C01806=1141.439,9.423,-49.221,179.746,6.279,149.212
C01807=1141.445,9.174,-49.208,179.743,6.278,149.213
C01808=1141.450,8.924,-49.194,179.741,6.277,149.213
C01809=1141.455,8.675,-49.181,179.739,6.276,149.214
C01810=1141.460,8.425,-49.167,179.736,6.275,149.214
C01811=1141.465,8.175,-49.153,179.733,6.274,149.215
C01812=1141.470,7.926,-49.140,179.731,6.273,149.215
C01813=1141.475,7.676,-49.126,179.729,6.273,149.216
C01814=1141.480,7.427,-49.113,179.726,6.272,149.216
C01815=1141.485,7.177,-49.100,179.723,6.271,149.217
C01816=1141.491,6.928,-49.086,179.721,6.270,149.217
C01817=1141.495,6.678,-49.073,179.718,6.269,149.218
C01818=1141.501,6.429,-49.059,179.716,6.269,149.219
C01819=1141.506,6.178,-49.045,179.714,6.268,149.219
C01820=1141.511,5.929,-49.033,179.711,6.266,149.220
C01821=1141.516,5.679,-49.018,179.709,6.266,149.220
C01822=1141.522,5.430,-49.006,179.706,6.265,149.221
C01823=1141.526,5.180,-48.991,179.704,6.264,149.221
C01824=1141.532,4.931,-48.979,179.701,6.263,149.222
C01825=1141.537,4.681,-48.965,179.698,6.262,149.223
C01826=1141.542,4.432,-48.951,179.696,6.262,149.223
C01827=1141.547,4.182,-48.938,179.693,6.261,149.224
C01828=1141.552,3.933,-48.924,179.691,6.260,149.224
C01829=1141.557,3.683,-48.911,179.689,6.259,149.225
C01830=1141.563,3.433,-48.898,179.686,6.258,149.225
C01831=1141.568,3.184,-48.885,179.684,6.257,149.226
C01832=1141.573,2.934,-48.871,179.681,6.257,149.226
C01833=1141.578,2.685,-48.859,179.678,6.255,149.227
C01834=1141.583,2.435,-48.845,179.676,6.255,149.227
C01835=1141.588,2.186,-48.832,179.673,6.254,149.228
C01836=1141.593,1.935,-48.818,179.671,6.253,149.228
C01837=1141.599,1.667,-48.804,179.668,6.252,149.229
C01838=1141.604,1.397,-48.790,179.666,6.251,149.230
C01839=1141.610,1.127,-48.776,179.663,6.251,149.230
C01840=1141.615,0.858,-48.762,179.660,6.249,149.231
C01841=1141.621,0.608,-48.748,179.658,6.249,149.231
C01842=1141.626,0.359,-48.736,179.656,6.248,149.232
C01843=1141.631,0.109,-48.721,179.653,6.248,149.233
C01844=1141.636,-0.140,-48.709,179.650,6.246,149.233
C01845=1141.642,-0.390,-48.696,179.648,6.245,149.234
C01846=1141.646,-0.640,-48.683,179.645,6.245,149.234
C01847=1141.651,-0.889,-48.670,179.643,6.244,149.235
C01848=1141.656,-1.139,-48.656,179.640,6.244,149.235
C01849=1141.662,-1.388,-48.643,179.638,6.243,149.236
C01850=1141.667,-1.638,-48.630,179.635,6.241,149.236
C01851=1141.672,-1.888,-48.617,179.633,6.241,149.237
C01852=1141.678,-2.138,-48.604,179.631,6.240,149.238
C01853=1141.683,-2.387,-48.591,179.628,6.240,149.238
C01854=1141.687,-2.637,-48.578,179.626,6.239,149.239
C01855=1141.693,-2.886,-48.564,179.623,6.237,149.239
C01856=1141.698,-3.135,-48.552,179.620,6.237,149.240
C01857=1141.703,-3.385,-48.539,179.618,6.236,149.240
C01858=1141.708,-3.635,-48.525,179.616,6.235,149.241
C01859=1141.713,-3.885,-48.513,179.613,6.235,149.241
C01860=1141.718,-4.134,-48.500,179.611,6.234,149.242
C01861=1141.724,-4.384,-48.487,179.608,6.233,149.243
C01862=1141.729,-4.634,-48.474,179.606,6.232,149.243
C01863=1141.734,-4.883,-48.461,179.603,6.231,149.244
C01864=1141.739,-5.133,-48.448,179.601,6.231,149.244
C01865=1141.745,-5.382,-48.435,179.599,6.230,149.245
C01866=1141.749,-5.632,-48.422,179.596,6.229,149.245
C01867=1141.755,-5.882,-48.409,179.593,6.228,149.246
C01868=1141.760,-6.131,-48.397,179.591,6.227,149.247
C01869=1141.765,-6.381,-48.384,179.588,6.227,149.247
C01870=1141.771,-6.631,-48.370,179.586,6.226,149.247
C01871=1141.776,-6.880,-48.358,179.584,6.225,149.248
C01872=1141.780,-7.130,-48.345,179.581,6.225,149.249
C01873=1141.785,-7.379,-48.332,179.579,6.224,149.249
C01874=1141.791,-7.629,-48.319,179.576,6.223,149.250
C01875=1141.796,-7.878,-48.306,179.574,6.222,149.250
C01876=1141.801,-8.128,-48.293,179.571,6.221,149.251
C01877=1141.806,-8.378,-48.281,179.569,6.220,149.251
C01878=1141.812,-8.627,-48.268,179.566,6.220,149.252
C01879=1141.817,-8.877,-48.255,179.564,6.219,149.253
C01880=1141.821,-9.127,-48.242,179.562,6.218,149.253
C01881=1141.827,-9.376,-48.230,179.559,6.217,149.254
C01882=1141.832,-9.625,-48.217,179.557,6.216,149.254
C01883=1141.838,-9.875,-48.204,179.554,6.216,149.255
C01884=1141.842,-10.126,-48.191,179.552,6.215,149.255
C01885=1141.847,-10.375,-48.179,179.550,6.214,149.256
C01886=1141.853,-10.624,-48.166,179.547,6.214,149.257
C01887=1141.858,-10.874,-48.154,179.545,6.213,149.257
C01888=1141.863,-11.124,-48.140,179.542,6.213,149.258
C01889=1141.868,-11.373,-48.128,179.539,6.211,149.258
C01890=1141.873,-11.623,-48.115,179.537,6.210,149.259
C01891=1141.879,-11.872,-48.103,179.534,6.210,149.259
C01892=1141.884,-12.122,-48.090,179.532,6.209,149.260
C01893=1141.888,-12.372,-48.077,179.530,6.209,149.260
C01894=1141.893,-12.621,-48.065,179.527,6.208,149.261
C01895=1141.899,-12.871,-48.052,179.525,6.207,149.261
C01896=1141.905,-13.121,-48.040,179.523,6.207,149.262
C01897=1141.910,-13.370,-48.027,179.520,6.205,149.263
C01898=1141.914,-13.620,-48.014,179.517,6.205,149.263
C01899=1141.920,-13.869,-48.002,179.515,6.204,149.264
C01900=1141.925,-14.119,-47.990,179.513,6.203,149.264
C01901=1141.930,-14.369,-47.977,179.510,6.203,149.265
C01902=1141.935,-14.618,-47.965,179.508,6.202,149.265
C01903=1141.940,-14.868,-47.952,179.506,6.201,149.266
C01904=1141.946,-15.118,-47.939,179.503,6.201,149.267
C01905=1141.951,-15.368,-47.926,179.501,6.200,149.267
C01906=1141.956,-15.617,-47.914,179.498,6.199,149.268
C01907=1141.962,-15.867,-47.902,179.495,6.198,149.268
C01908=1141.967,-16.116,-47.889,179.493,6.197,149.269
C01909=1141.972,-16.365,-47.877,179.491,6.197,149.269
C01910=1141.977,-16.616,-47.865,179.488,6.196,149.270
C01911=1141.982,-16.865,-47.852,179.486,6.195,149.270
C01912=1141.987,-17.115,-47.839,179.484,6.195,149.271
C01913=1141.992,-17.365,-47.827,179.481,6.194,149.271
C01914=1141.997,-17.614,-47.815,179.479,6.193,149.272
C01915=1142.003,-17.864,-47.803,179.477,6.193,149.273
C01916=1142.008,-18.113,-47.790,179.474,6.192,149.273
C01917=1142.013,-18.362,-47.778,179.472,6.191,149.274
C01918=1142.019,-18.612,-47.766,179.470,6.191,149.274
C01919=1142.023,-18.862,-47.753,179.466,6.189,149.275
C01920=1142.028,-19.112,-47.741,179.464,6.189,149.275
C01921=1142.034,-19.362,-47.728,179.461,6.188,149.276
C01922=1142.039,-19.611,-47.716,179.459,6.187,149.277
C01923=1142.044,-19.861,-47.704,179.457,6.187,149.277
C01924=1142.049,-20.110,-47.691,179.454,6.186,149.278
C01925=1142.055,-20.360,-47.679,179.452,6.185,149.278
C01926=1142.060,-20.610,-47.667,179.450,6.185,149.279
C01927=1142.065,-20.859,-47.655,179.447,6.184,149.279
C01928=1142.070,-21.109,-47.642,179.445,6.183,149.280
C01929=1142.076,-21.359,-47.630,179.443,6.183,149.281
C01930=1142.081,-21.608,-47.618,179.440,6.182,149.281
C01931=1142.086,-21.858,-47.606,179.438,6.181,149.281
C01932=1142.091,-22.107,-47.593,179.436,6.181,149.282
C01933=1142.097,-22.357,-47.582,179.433,6.180,149.283
C01934=1142.101,-22.606,-47.570,179.431,6.180,149.283
C01935=1142.106,-22.857,-47.557,179.428,6.178,149.284
C01936=1142.111,-23.106,-47.545,179.426,6.177,149.284
C01937=1142.117,-23.356,-47.533,179.423,6.177,149.285
C01938=1142.122,-23.606,-47.521,179.421,6.176,149.285
C01939=1142.127,-23.855,-47.508,179.418,6.176,149.286
C01940=1142.133,-24.105,-47.496,179.416,6.175,149.287
C01941=1142.139,-24.375,-47.484,179.413,6.175,149.287
C01942=1142.144,-24.645,-47.470,179.411,6.174,149.288
C01943=1142.149,-24.915,-47.457,179.409,6.173,149.288
C01944=1142.156,-25.185,-47.444,179.406,6.172,149.289
C01945=1142.160,-25.435,-47.433,179.403,6.171,149.290
C01946=1142.165,-25.684,-47.420,179.401,6.171,149.290
C01947=1142.171,-25.934,-47.408,179.399,6.170,149.291
C01948=1142.176,-26.184,-47.396,179.396,6.169,149.291
C01949=1142.181,-26.433,-47.384,179.394,6.169,149.292
C01950=1142.186,-26.683,-47.372,179.391,6.168,149.292
C01951=1142.191,-26.933,-47.361,179.389,6.167,149.293
C01952=1142.197,-27.182,-47.348,179.387,6.167,149.293
C01953=1142.202,-27.432,-47.336,179.384,6.166,149.294
C01954=1142.207,-27.682,-47.324,179.382,6.165,149.295
C01955=1142.212,-27.931,-47.312,179.380,6.165,149.295
C01956=1142.217,-28.181,-47.300,179.377,6.164,149.296
C01957=1142.223,-28.431,-47.288,179.375,6.163,149.296
C01958=1142.228,-28.681,-47.276,179.372,6.163,149.297
C01959=1142.233,-28.930,-47.264,179.370,6.162,149.297
C01960=1142.238,-29.180,-47.253,179.368,6.161,149.298
C01961=1142.243,-29.430,-47.241,179.365,6.161,149.299
C01962=1142.249,-29.680,-47.229,179.363,6.160,149.299
C01963=1142.254,-29.928,-47.217,179.360,6.160,149.300
C01964=1142.259,-30.178,-47.205,179.358,6.159,149.300
C01965=1142.265,-30.428,-47.193,179.356,6.158,149.301
C01966=1142.270,-30.678,-47.182,179.353,6.158,149.301
C01967=1142.275,-30.927,-47.170,179.351,6.157,149.302
C01968=1142.280,-31.177,-47.158,179.349,6.156,149.302
C01969=1142.285,-31.427,-47.146,179.346,6.156,149.303
C01970=1142.290,-31.676,-47.134,179.344,6.155,149.304
C01971=1142.295,-31.926,-47.123,179.342,6.155,149.304
C01972=1142.301,-32.176,-47.111,179.339,6.154,149.305
C01973=1142.306,-32.425,-47.098,179.337,6.153,149.305
C01974=1142.311,-32.674,-47.087,179.334,6.153,149.306
C01975=1142.317,-32.924,-47.075,179.332,6.152,149.306
C01976=1142.322,-33.174,-47.063,179.330,6.151,149.307
C01977=1142.327,-33.424,-47.052,179.327,6.151,149.308
C01978=1142.332,-33.674,-47.040,179.325,6.150,149.308
C01979=1142.338,-33.924,-47.028,179.323,6.150,149.309
C01980=1142.342,-34.173,-47.017,179.320,6.149,149.309
C01981=1142.348,-34.423,-47.005,179.318,6.148,149.310
C01982=1142.353,-34.672,-46.994,179.316,6.148,149.310
C01983=1142.358,-34.921,-46.982,179.313,6.147,149.311
C01984=1142.364,-35.171,-46.970,179.311,6.146,149.311
C01985=1142.368,-35.421,-46.958,179.309,6.146,149.312
C01986=1142.374,-35.671,-46.947,179.306,6.145,149.312
C01987=1142.379,-35.921,-46.935,179.304,6.144,149.313
C01988=1142.385,-36.170,-46.924,179.301,6.144,149.314
C01989=1142.390,-36.420,-46.912,179.299,6.143,149.314
C01990=1142.395,-36.669,-46.901,179.297,6.142,149.315
C01991=1142.400,-36.919,-46.889,179.294,6.142,149.315
C01992=1142.405,-37.169,-46.877,179.292,6.141,149.316
C01993=1142.411,-37.418,-46.866,179.290,6.140,149.316
C01994=1142.416,-37.668,-46.854,179.288,6.140,149.317
C01995=1142.421,-37.918,-46.843,179.286,6.140,149.317
C01996=1142.426,-38.168,-46.831,179.283,6.139,149.318
C01997=1142.431,-38.417,-46.820,179.281,6.138,149.319
C01998=1142.437,-38.667,-46.808,179.278,6.138,149.319
C01999=1142.442,-38.916,-46.797,179.276,6.137,149.320
C02000=1142.447,-39.167,-46.786,179.274,6.136,149.320
C02001=1142.453,-39.417,-46.774,179.271,6.136,149.321
C02002=1142.458,-39.666,-46.762,179.269,6.135,149.321
C02003=1142.464,-39.915,-46.751,179.267,6.135,149.322
C02004=1142.468,-40.165,-46.740,179.264,6.134,149.323
C02005=1142.474,-40.415,-46.728,179.262,6.133,149.323
C02006=1142.478,-40.665,-46.716,179.260,6.133,149.324
C02007=1142.484,-40.914,-46.705,179.257,6.132,149.324
C02008=1142.489,-41.164,-46.694,179.255,6.131,149.325
C02009=1142.495,-41.413,-46.682,179.252,6.131,149.325
C02010=1142.500,-41.664,-46.671,179.250,6.130,149.326
C02011=1142.506,-41.913,-46.660,179.248,6.129,149.326
C02012=1142.510,-42.163,-46.648,179.245,6.129,149.327
C02013=1142.515,-42.412,-46.637,179.244,6.129,149.328
C02014=1142.520,-42.662,-46.625,179.242,6.128,149.328
C02015=1142.526,-42.911,-46.614,179.239,6.128,149.329
C02016=1142.531,-43.162,-46.603,179.237,6.127,149.329
C02017=1142.536,-43.411,-46.592,179.235,6.126,149.330
C02018=1142.542,-43.661,-46.580,179.232,6.126,149.330
C02019=1142.547,-43.910,-46.569,179.230,6.125,149.331
C02020=1142.552,-44.160,-46.558,179.227,6.124,149.331
C02021=1142.557,-44.410,-46.547,179.225,6.124,149.332
C02022=1142.563,-44.659,-46.536,179.223,6.123,149.333
C02023=1142.568,-44.909,-46.524,179.220,6.123,149.333
C02024=1142.573,-45.159,-46.512,179.218,6.122,149.334
C02025=1142.578,-45.408,-46.502,179.216,6.121,149.334
C02026=1142.584,-45.658,-46.490,179.213,6.122,149.335
C02027=1142.588,-45.908,-46.479,179.211,6.121,149.335
C02028=1142.594,-46.158,-46.467,179.209,6.120,149.336
C02029=1142.599,-46.407,-46.457,179.206,6.120,149.337
C02030=1142.604,-46.657,-46.446,179.204,6.119,149.337
C02031=1142.610,-46.907,-46.434,179.202,6.118,149.337
C02032=1142.615,-47.156,-46.424,179.199,6.118,149.338
C02033=1142.620,-47.406,-46.412,179.197,6.117,149.339
C02034=1142.625,-47.656,-46.400,179.195,6.116,149.339
C02035=1142.631,-47.906,-46.390,179.192,6.116,149.340
C02036=1142.636,-48.155,-46.379,179.190,6.115,149.340
C02037=1142.642,-48.404,-46.367,179.189,6.115,149.341
C02038=1142.647,-48.655,-46.357,179.186,6.115,149.341
C02039=1142.651,-48.904,-46.345,179.184,6.114,149.342
C02040=1142.657,-49.154,-46.334,179.182,6.113,149.342
C02041=1142.662,-49.404,-46.323,179.179,6.113,149.343
C02042=1142.667,-49.653,-46.312,179.177,6.112,149.344
C02043=1142.673,-49.903,-46.301,179.174,6.111,149.344
C02044=1142.678,-50.153,-46.290,179.172,6.111,149.345
C02045=1142.684,-50.424,-46.278,179.170,6.110,149.345
C02046=1142.690,-50.694,-46.266,179.167,6.109,149.346
C02047=1142.695,-50.965,-46.254,179.165,6.109,149.346
C02048=1142.701,-51.235,-46.242,179.162,6.108,149.347
C02049=1142.706,-51.485,-46.232,179.160,6.108,149.348
C02050=1142.711,-51.735,-46.220,179.157,6.107,149.348
C02051=1142.717,-51.985,-46.210,179.155,6.106,149.349
C02052=1142.722,-52.234,-46.198,179.153,6.106,149.349
C02053=1142.727,-52.484,-46.188,179.151,6.106,149.350
C02054=1142.733,-52.734,-46.176,179.149,6.105,149.351
C02055=1142.738,-52.984,-46.166,179.146,6.104,149.351
C02056=1142.743,-53.233,-46.155,179.144,6.104,149.352
C02057=1142.748,-53.483,-46.144,179.142,6.103,149.352
C02058=1142.753,-53.732,-46.133,179.139,6.102,149.353
C02059=1142.759,-53.983,-46.122,179.137,6.103,149.353
C02060=1142.764,-54.232,-46.111,179.135,6.102,149.354
C02061=1142.769,-54.482,-46.101,179.133,6.101,149.354
C02062=1142.774,-54.732,-46.089,179.130,6.101,149.355
C02063=1142.780,-54.981,-46.079,179.128,6.100,149.355
C02064=1142.785,-55.231,-46.067,179.126,6.099,149.356
C02065=1142.791,-55.481,-46.057,179.123,6.099,149.357
C02066=1142.795,-55.730,-46.046,179.121,6.098,149.357
C02067=1142.801,-55.980,-46.036,179.119,6.098,149.358
C02068=1142.806,-56.230,-46.025,179.117,6.098,149.358
C02069=1142.811,-56.479,-46.014,179.115,6.097,149.359
C02070=1142.816,-56.729,-46.003,179.112,6.096,149.359
C02071=1142.822,-56.978,-45.992,179.110,6.096,149.360
C02072=1142.827,-57.229,-45.981,179.108,6.095,149.360
C02073=1142.832,-57.479,-45.971,179.106,6.095,149.361
C02074=1142.838,-57.728,-45.960,179.103,6.095,149.362
C02075=1142.843,-57.978,-45.949,179.101,6.094,149.362
C02076=1142.848,-58.228,-45.939,179.099,6.093,149.363
C02077=1142.853,-58.477,-45.928,179.096,6.093,149.363
C02078=1142.858,-58.727,-45.918,179.094,6.092,149.364
C02079=1142.863,-58.976,-45.906,179.092,6.091,149.364
C02080=1142.869,-59.226,-45.895,179.090,6.091,149.365
C02081=1142.874,-59.477,-45.885,179.088,6.091,149.365
C02082=1142.880,-59.726,-45.875,179.085,6.090,149.366
C02083=1142.885,-59.976,-45.863,179.083,6.089,149.366
C02084=1142.890,-60.225,-45.853,179.081,6.089,149.367
C02085=1142.895,-60.476,-45.843,179.078,6.088,149.368
C02086=1142.901,-60.724,-45.832,179.077,6.088,149.368
C02087=1142.906,-60.974,-45.821,179.074,6.088,149.369
C02088=1142.911,-61.224,-45.811,179.072,6.087,149.369
C02089=1142.917,-61.474,-45.801,179.070,6.086,149.370
C02090=1142.922,-61.723,-45.789,179.067,6.086,149.370
C02091=1142.927,-61.973,-45.779,179.065,6.085,149.371
C02092=1142.932,-62.223,-45.769,179.063,6.085,149.371
C02093=1142.938,-62.473,-45.758,179.061,6.085,149.372
C02094=1142.942,-62.722,-45.747,179.058,6.084,149.373
C02095=1142.948,-62.972,-45.737,179.056,6.083,149.373
C02096=1142.953,-63.222,-45.726,179.054,6.082,149.374
C02097=1142.959,-63.472,-45.716,179.052,6.083,149.374
C02098=1142.964,-63.721,-45.706,179.050,6.082,149.375
C02099=1142.969,-63.971,-45.695,179.048,6.081,149.375
C02100=1142.975,-64.220,-45.684,179.045,6.081,149.376
C02101=1142.980,-64.471,-45.674,179.043,6.080,149.376
C02102=1142.985,-64.720,-45.664,179.041,6.080,149.377
C02103=1142.991,-64.970,-45.653,179.038,6.080,149.378
C02104=1142.995,-65.219,-45.642,179.036,6.079,149.378
C02105=1143.001,-65.469,-45.632,179.034,6.078,149.379
C02106=1143.006,-65.719,-45.621,179.031,6.078,149.379
C02107=1143.012,-65.969,-45.611,179.030,6.078,149.380
C02108=1143.017,-66.218,-45.601,179.028,6.077,149.380
C02109=1143.022,-66.468,-45.590,179.025,6.076,149.381
C02110=1143.028,-66.718,-45.580,179.023,6.076,149.381
C02111=1143.033,-66.968,-45.570,179.021,6.075,149.382
C02112=1143.038,-67.218,-45.559,179.019,6.075,149.382
C02113=1143.044,-67.467,-45.548,179.016,6.075,149.383
C02114=1143.049,-67.717,-45.538,179.014,6.074,149.384
C02115=1143.054,-67.966,-45.528,179.012,6.073,149.384
C02116=1143.059,-68.216,-45.518,179.010,6.073,149.385
C02117=1143.064,-68.466,-45.507,179.008,6.073,149.385
C02118=1143.070,-68.716,-45.497,179.005,6.072,149.386
C02119=1143.075,-68.966,-45.487,179.003,6.071,149.386
C02120=1143.080,-69.215,-45.477,179.001,6.071,149.387
C02121=1143.086,-69.465,-45.466,178.998,6.070,149.387
C02122=1143.091,-69.715,-45.456,178.997,6.070,149.388
C02123=1143.097,-69.965,-45.446,178.995,6.070,149.388
C02124=1143.101,-70.214,-45.436,178.992,6.069,149.389
C02125=1143.106,-70.464,-45.425,178.990,6.068,149.390
C02126=1143.112,-70.714,-45.415,178.988,6.068,149.390
C02127=1143.118,-70.963,-45.405,178.985,6.068,149.391
C02128=1143.123,-71.213,-45.394,178.983,6.067,149.391
C02129=1143.128,-71.463,-45.384,178.981,6.066,149.392
C02130=1143.134,-71.713,-45.374,178.979,6.066,149.392
C02131=1143.139,-71.962,-45.364,178.977,6.066,149.393
C02132=1143.144,-72.212,-45.354,178.975,6.065,149.393
C02133=1143.149,-72.462,-45.344,178.972,6.065,149.394
C02134=1143.155,-72.711,-45.333,178.970,6.064,149.395
C02135=1143.160,-72.961,-45.323,178.968,6.064,149.395
C02136=1143.166,-73.212,-45.313,178.966,6.063,149.396
C02137=1143.171,-73.461,-45.304,178.964,6.063,149.396
C02138=1143.176,-73.711,-45.293,178.961,6.062,149.397
C02139=1143.181,-73.961,-45.283,178.960,6.062,149.397
C02140=1143.187,-74.210,-45.273,178.957,6.062,149.398
C02141=1143.192,-74.460,-45.262,178.955,6.061,149.398
C02142=1143.197,-74.710,-45.252,178.952,6.060,149.399
C02143=1143.202,-74.959,-45.242,178.951,6.060,149.399
C02144=1143.208,-75.209,-45.232,178.949,6.060,149.400
C02145=1143.214,-75.459,-45.223,178.946,6.059,149.401
C02146=1143.218,-75.709,-45.213,178.944,6.059,149.401
C02147=1143.224,-75.958,-45.202,178.942,6.059,149.402
C02148=1143.229,-76.208,-45.192,178.940,6.058,149.402
C02149=1143.234,-76.479,-45.181,178.937,6.057,149.403
C02150=1143.241,-76.751,-45.170,178.935,6.057,149.403
C02151=1143.246,-77.022,-45.160,178.933,6.056,149.404
C02152=1143.252,-77.294,-45.148,178.930,6.056,149.404
C02153=1143.257,-77.543,-45.139,178.928,6.055,149.405
C02154=1143.263,-77.793,-45.129,178.926,6.055,149.406
C02155=1143.268,-78.043,-45.119,178.924,6.054,149.406
C02156=1143.274,-78.293,-45.108,178.922,6.054,149.407
C02157=1143.279,-78.542,-45.099,178.920,6.054,149.407
C02158=1143.284,-78.792,-45.089,178.917,6.053,149.408
C02159=1143.290,-79.042,-45.079,178.915,6.053,149.408
C02160=1143.294,-79.292,-45.069,178.913,6.052,149.409
C02161=1143.300,-79.541,-45.059,178.911,6.052,149.409
C02162=1143.306,-79.791,-45.049,178.909,6.051,149.410
C02163=1143.311,-80.041,-45.040,178.907,6.051,149.410
C02164=1143.316,-80.290,-45.030,178.904,6.050,149.411
C02165=1143.322,-80.541,-45.020,178.902,6.050,149.412
C02166=1143.326,-80.790,-45.010,178.900,6.050,149.412
C02167=1143.332,-81.040,-45.000,178.898,6.049,149.413
C02168=1143.338,-81.289,-44.990,178.896,6.049,149.413
C02169=1143.343,-81.539,-44.981,178.894,6.048,149.414
C02170=1143.348,-81.789,-44.970,178.891,6.048,149.414
C02171=1143.353,-82.039,-44.961,178.889,6.047,149.415
C02172=1143.359,-82.289,-44.951,178.888,6.047,149.415
C02173=1143.364,-82.538,-44.941,178.885,6.046,149.416
C02174=1143.369,-82.788,-44.931,178.883,6.046,149.416
C02175=1143.375,-83.038,-44.922,178.881,6.046,149.417
C02176=1143.381,-83.287,-44.912,178.879,6.045,149.417
C02177=1143.385,-83.537,-44.902,178.877,6.044,149.418
C02178=1143.391,-83.787,-44.892,178.874,6.044,149.419
C02179=1143.396,-84.037,-44.882,178.873,6.044,149.419
C02180=1143.401,-84.287,-44.873,178.870,6.043,149.419
C02181=1143.406,-84.536,-44.863,178.868,6.042,149.420
C02182=1143.412,-84.786,-44.853,178.866,6.043,149.421
C02183=1143.417,-85.036,-44.843,178.864,6.042,149.421
C02184=1143.422,-85.286,-44.834,178.862,6.041,149.422
C02185=1143.428,-85.536,-44.824,178.859,6.041,149.422
C02186=1143.433,-85.785,-44.815,178.857,6.041,149.423
C02187=1143.439,-86.035,-44.805,178.855,6.040,149.423
C02188=1143.444,-86.284,-44.795,178.853,6.040,149.424
C02189=1143.449,-86.534,-44.785,178.851,6.040,149.424
C02190=1143.454,-86.784,-44.776,178.849,6.039,149.425
C02191=1143.460,-87.033,-44.766,178.847,6.038,149.425
C02192=1143.465,-87.284,-44.757,178.845,6.038,149.426
C02193=1143.470,-87.533,-44.747,178.843,6.038,149.426
C02194=1143.475,-87.783,-44.738,178.841,6.037,149.427
C02195=1143.481,-88.033,-44.728,178.839,6.037,149.428
C02196=1143.486,-88.283,-44.719,178.836,6.037,149.428
C02197=1143.492,-88.532,-44.708,178.834,6.036,149.429
C02198=1143.497,-88.782,-44.700,178.832,6.035,149.429
C02199=1143.502,-89.032,-44.689,178.830,6.035,149.430
C02200=1143.508,-89.281,-44.680,178.828,6.035,149.430
C02201=1143.513,-89.531,-44.670,178.825,6.034,149.431
C02202=1143.518,-89.781,-44.661,178.824,6.034,149.431
C02203=1143.523,-90.031,-44.651,178.822,6.033,149.432
C02204=1143.529,-90.281,-44.642,178.819,6.032,149.432
C02205=1143.534,-90.531,-44.632,178.817,6.033,149.433
C02206=1143.539,-90.780,-44.623,178.815,6.032,149.433
C02207=1143.545,-91.031,-44.613,178.813,6.031,149.434
C02208=1143.550,-91.280,-44.604,178.811,6.031,149.434
C02209=1143.555,-91.530,-44.595,178.809,6.031,149.435
C02210=1143.561,-91.779,-44.585,178.807,6.030,149.436
C02211=1143.566,-92.029,-44.576,178.805,6.030,149.436
C02212=1143.572,-92.279,-44.566,178.803,6.030,149.437
C02213=1143.577,-92.528,-44.557,178.801,6.029,149.437
C02214=1143.583,-92.779,-44.547,178.799,6.029,149.438
C02215=1143.588,-93.028,-44.538,178.796,6.028,149.438
C02216=1143.593,-93.278,-44.529,178.794,6.028,149.439
C02217=1143.599,-93.528,-44.519,178.793,6.028,149.439
C02218=1143.603,-93.777,-44.509,178.790,6.027,149.440
C02219=1143.609,-94.027,-44.501,178.788,6.026,149.440
C02220=1143.615,-94.277,-44.491,178.786,6.027,149.441
C02221=1143.619,-94.526,-44.481,178.784,6.026,149.441
C02222=1143.625,-94.776,-44.472,178.782,6.025,149.442
C02223=1143.630,-95.026,-44.463,178.780,6.025,149.442
C02224=1143.635,-95.276,-44.453,178.778,6.024,149.443
C02225=1143.641,-95.526,-44.444,178.776,6.025,149.444
C02226=1143.646,-95.776,-44.435,178.774,6.024,149.444
C02227=1143.652,-96.025,-44.426,178.771,6.023,149.445
C02228=1143.657,-96.275,-44.416,178.770,6.023,149.445
C02229=1143.662,-96.525,-44.407,178.768,6.023,149.445
C02230=1143.667,-96.775,-44.398,178.765,6.022,149.446
C02231=1143.673,-97.025,-44.389,178.763,6.022,149.447
C02232=1143.678,-97.274,-44.379,178.761,6.022,149.447
C02233=1143.683,-97.524,-44.370,178.759,6.021,149.448
C02234=1143.689,-97.774,-44.361,178.757,6.021,149.448
C02235=1143.694,-98.024,-44.352,178.755,6.020,149.449
C02236=1143.699,-98.273,-44.342,178.752,6.020,149.449
C02237=1143.705,-98.523,-44.333,178.751,6.020,149.450
C02238=1143.710,-98.773,-44.324,178.749,6.019,149.450
C02239=1143.716,-99.023,-44.315,178.747,6.019,149.451
C02240=1143.721,-99.273,-44.305,178.745,6.018,149.451
C02241=1143.727,-99.522,-44.296,178.743,6.017,149.452
C02242=1143.732,-99.772,-44.287,178.741,6.018,149.452
C02243=1143.737,-100.021,-44.278,178.738,6.017,149.453
C02244=1143.743,-100.272,-44.269,178.736,6.016,149.453
C02245=1143.748,-100.521,-44.260,178.735,6.016,149.454
C02246=1143.753,-100.771,-44.250,178.732,6.016,149.454
C02247=1143.759,-101.021,-44.241,178.731,6.016,149.455
C02248=1143.764,-101.271,-44.232,178.728,6.015,149.456
C02249=1143.769,-101.520,-44.223,178.726,6.015,149.456
C02250=1143.775,-101.770,-44.214,178.724,6.015,149.457
C02251=1143.780,-102.020,-44.205,178.722,6.014,149.457
C02252=1143.785,-102.270,-44.195,178.720,6.013,149.458
C02253=1143.792,-102.542,-44.186,178.718,6.014,149.458
C02254=1143.797,-102.813,-44.176,178.716,6.013,149.459
C02255=1143.803,-103.086,-44.166,178.714,6.012,149.459
C02256=1143.809,-103.358,-44.156,178.711,6.012,149.460
C02257=1143.814,-103.608,-44.147,178.709,6.012,149.460
C02258=1143.820,-103.858,-44.138,178.707,6.011,149.461
C02259=1143.825,-104.108,-44.129,178.705,6.011,149.461
C02260=1143.830,-104.358,-44.120,178.703,6.010,149.462
C02261=1143.836,-104.607,-44.111,178.701,6.010,149.462
C02262=1143.841,-104.857,-44.102,178.699,6.010,149.463
C02263=1143.846,-105.107,-44.093,178.697,6.009,149.464
C02264=1143.852,-105.357,-44.084,178.695,6.009,149.464
C02265=1143.857,-105.607,-44.075,178.693,6.008,149.465
C02266=1143.862,-105.856,-44.066,178.691,6.008,149.465
C02267=1143.867,-106.106,-44.057,178.689,6.008,149.466
C02268=1143.873,-106.355,-44.049,178.687,6.007,149.466
C02269=1143.878,-106.605,-44.040,178.685,6.007,149.467
C02270=1143.884,-106.855,-44.031,178.683,6.007,149.467
C02271=1143.889,-107.105,-44.021,178.681,6.006,149.468
C02272=1143.895,-107.355,-44.012,178.679,6.006,149.468
C02273=1143.900,-107.605,-44.004,178.677,6.005,149.469
C02274=1143.906,-107.854,-43.995,178.675,6.005,149.469
C02275=1143.911,-108.104,-43.986,178.673,6.005,149.470
C02276=1143.916,-108.354,-43.977,178.671,6.004,149.470
C02277=1143.921,-108.604,-43.968,178.669,6.004,149.471
C02278=1143.926,-108.854,-43.959,178.666,6.003,149.471
C02279=1143.932,-109.104,-43.950,178.665,6.003,149.472
C02280=1143.938,-109.353,-43.941,178.663,6.003,149.472
C02281=1143.943,-109.603,-43.933,178.660,6.002,149.473
C02282=1143.948,-109.853,-43.924,178.659,6.002,149.473
C02283=1143.953,-110.102,-43.915,178.657,6.001,149.474
C02284=1143.959,-110.352,-43.906,178.655,6.001,149.474
C02285=1143.964,-110.601,-43.897,178.653,6.001,149.475
C02286=1143.970,-110.852,-43.889,178.651,6.001,149.475
C02287=1143.975,-111.102,-43.880,178.649,6.000,149.476
C02288=1143.980,-111.352,-43.871,178.646,6.000,149.476
C02289=1143.985,-111.601,-43.862,178.645,6.000,149.477
C02290=1143.991,-111.851,-43.854,178.643,5.999,149.477
C02291=1143.996,-112.100,-43.845,178.641,5.999,149.478
C02292=1144.001,-112.350,-43.836,178.639,5.998,149.478
C02293=1144.007,-112.600,-43.827,178.637,5.998,149.479
C02294=1144.013,-112.850,-43.819,178.635,5.997,149.479
C02295=1144.019,-113.100,-43.810,178.632,5.997,149.480
C02296=1144.024,-113.350,-43.801,178.631,5.997,149.481
C02297=1144.029,-113.600,-43.792,178.629,5.996,149.481
C02298=1144.035,-113.849,-43.784,178.627,5.996,149.482
C02299=1144.040,-114.099,-43.775,178.625,5.996,149.482
C02300=1144.045,-114.349,-43.767,178.623,5.996,149.482
C02301=1144.050,-114.599,-43.758,178.621,5.995,149.483
C02302=1144.056,-114.848,-43.749,178.619,5.994,149.483
C02303=1144.061,-115.098,-43.740,178.617,5.994,149.484
C02304=1144.067,-115.348,-43.731,178.615,5.993,149.484
C02305=1144.072,-115.598,-43.723,178.613,5.994,149.485
C02306=1144.078,-115.848,-43.715,178.611,5.993,149.486
C02307=1144.083,-116.097,-43.706,178.609,5.993,149.486
C02308=1144.088,-116.347,-43.697,178.607,5.992,149.487
C02309=1144.093,-116.597,-43.688,178.605,5.992,149.487
C02310=1144.099,-116.847,-43.681,178.603,5.992,149.488
C02311=1144.104,-117.096,-43.672,178.601,5.991,149.488
C02312=1144.109,-117.346,-43.663,178.599,5.991,149.489
C02313=1144.115,-117.596,-43.655,178.597,5.990,149.489
C02314=1144.120,-117.846,-43.646,178.596,5.990,149.490
C02315=1144.125,-118.096,-43.637,178.593,5.990,149.490
C02316=1144.131,-118.345,-43.629,178.592,5.990,149.491
C02317=1144.137,-118.595,-43.621,178.590,5.989,149.491
C02318=1144.142,-118.845,-43.612,178.588,5.989,149.492
C02319=1144.147,-119.095,-43.603,178.585,5.989,149.492
C02320=1144.153,-119.345,-43.595,178.584,5.989,149.493
C02321=1144.158,-119.595,-43.586,178.582,5.988,149.493
C02322=1144.163,-119.845,-43.577,178.580,5.988,149.494
C02323=1144.169,-120.094,-43.569,178.578,5.987,149.494
C02324=1144.174,-120.344,-43.561,178.576,5.986,149.495
C02325=1144.179,-120.594,-43.552,178.574,5.986,149.495
C02326=1144.185,-120.843,-43.544,178.572,5.986,149.496
C02327=1144.190,-121.093,-43.535,178.570,5.986,149.496
C02328=1144.195,-121.343,-43.526,178.568,5.985,149.497
C02329=1144.201,-121.593,-43.519,178.566,5.985,149.497
C02330=1144.207,-121.843,-43.510,178.564,5.984,149.498
C02331=1144.212,-122.093,-43.501,178.563,5.984,149.498
C02332=1144.217,-122.342,-43.494,178.560,5.984,149.499
C02333=1144.222,-122.592,-43.485,178.559,5.984,149.499
C02334=1144.228,-122.842,-43.477,178.557,5.983,149.500
C02335=1144.234,-123.092,-43.468,178.554,5.983,149.500
C02336=1144.239,-123.341,-43.459,178.552,5.983,149.501
C02337=1144.244,-123.592,-43.451,178.551,5.983,149.501
C02338=1144.249,-123.841,-43.443,178.548,5.982,149.502
C02339=1144.255,-124.091,-43.435,178.547,5.982,149.502
C02340=1144.260,-124.340,-43.426,178.545,5.981,149.503
C02341=1144.266,-124.590,-43.417,178.543,5.981,149.503
C02342=1144.271,-124.841,-43.409,178.541,5.980,149.504
C02343=1144.277,-125.090,-43.401,178.539,5.980,149.504
C02344=1144.282,-125.340,-43.393,178.537,5.980,149.505
C02345=1144.287,-125.590,-43.384,178.535,5.979,149.505
C02346=1144.293,-125.840,-43.376,178.533,5.979,149.506
C02347=1144.298,-126.089,-43.367,178.531,5.978,149.506
C02348=1144.303,-126.339,-43.360,178.530,5.978,149.507
C02349=1144.309,-126.589,-43.351,178.527,5.978,149.507
C02350=1144.314,-126.839,-43.343,178.526,5.978,149.508
C02351=1144.320,-127.088,-43.335,178.524,5.977,149.508
C02352=1144.325,-127.339,-43.326,178.522,5.977,149.509
C02353=1144.330,-127.588,-43.319,178.520,5.976,149.509
C02354=1144.336,-127.838,-43.310,178.518,5.976,149.510
C02355=1144.341,-128.087,-43.302,178.516,5.975,149.510
C02356=1144.347,-128.338,-43.294,178.514,5.976,149.510
C02357=1143.926,-128.348,-43.337,178.510,5.979,149.512
C02358=1143.921,-128.099,-43.345,178.513,5.980,149.512
C02359=1143.915,-127.849,-43.353,178.514,5.980,149.511
C02360=1143.909,-127.600,-43.362,178.516,5.980,149.511
C02361=1143.904,-127.349,-43.370,178.518,5.980,149.510
C02362=1143.899,-127.099,-43.379,178.520,5.981,149.510
C02363=1143.893,-126.850,-43.386,178.522,5.981,149.509
C02364=1143.888,-126.600,-43.395,178.524,5.982,149.509
C02365=1143.882,-126.350,-43.403,178.526,5.982,149.508
C02366=1143.877,-126.101,-43.412,178.528,5.982,149.508
C02367=1143.872,-125.850,-43.419,178.529,5.982,149.507
C02368=1143.866,-125.601,-43.428,178.532,5.983,149.507
C02369=1143.861,-125.351,-43.436,178.533,5.983,149.506
C02370=1143.855,-125.102,-43.444,178.535,5.984,149.506
C02371=1143.850,-124.851,-43.453,178.537,5.984,149.505
C02372=1143.845,-124.602,-43.461,178.539,5.984,149.505
C02373=1143.839,-124.352,-43.469,178.541,5.984,149.505
C02374=1143.834,-124.102,-43.478,178.544,5.985,149.504
C02375=1143.828,-123.853,-43.486,178.546,5.985,149.503
C02376=1143.823,-123.602,-43.494,178.547,5.985,149.503
C02377=1143.818,-123.353,-43.503,178.550,5.986,149.502
C02378=1143.812,-123.103,-43.510,178.551,5.986,149.502
C02379=1143.807,-122.853,-43.519,178.553,5.987,149.501
C02380=1143.802,-122.603,-43.528,178.555,5.987,149.501
C02381=1143.796,-122.354,-43.536,178.557,5.988,149.500
C02382=1143.791,-122.104,-43.545,178.559,5.988,149.500
C02383=1143.785,-121.853,-43.553,178.561,5.988,149.499
C02384=1143.780,-121.604,-43.561,178.562,5.988,149.499
C02385=1143.775,-121.355,-43.570,178.565,5.989,149.498
C02386=1143.770,-121.104,-43.578,178.566,5.989,149.498
C02387=1143.764,-120.855,-43.587,178.568,5.990,149.497
C02388=1143.758,-120.604,-43.595,178.570,5.990,149.497
C02389=1143.753,-120.355,-43.604,178.572,5.990,149.496
C02390=1143.747,-120.105,-43.612,178.574,5.990,149.496
C02391=1143.742,-119.855,-43.621,178.576,5.991,149.495
C02392=1143.737,-119.605,-43.629,178.578,5.992,149.495
C02393=1143.732,-119.356,-43.637,178.580,5.992,149.495
C02394=1143.727,-119.106,-43.646,178.583,5.992,149.494
C02395=1143.721,-118.856,-43.654,178.584,5.992,149.493
C02396=1143.715,-118.607,-43.663,178.586,5.993,149.493
C02397=1143.710,-118.357,-43.672,178.588,5.993,149.492
C02398=1143.705,-118.107,-43.680,178.590,5.994,149.492
C02399=1143.699,-117.857,-43.689,178.592,5.994,149.491
C02400=1143.694,-117.608,-43.697,178.594,5.994,149.491
C02401=1143.689,-117.358,-43.706,178.596,5.994,149.490
C02402=1143.683,-117.107,-43.715,178.598,5.995,149.490
C02403=1143.677,-116.858,-43.723,178.600,5.996,149.489
C02404=1143.672,-116.608,-43.732,178.602,5.996,149.489
C02405=1143.667,-116.358,-43.740,178.604,5.996,149.488
C02406=1143.661,-116.109,-43.749,178.605,5.996,149.488
C02407=1143.656,-115.859,-43.758,178.608,5.997,149.487
C02408=1143.651,-115.609,-43.767,178.610,5.997,149.487
C02409=1143.645,-115.359,-43.775,178.612,5.997,149.486
C02410=1143.639,-115.109,-43.783,178.613,5.997,149.486
C02411=1143.634,-114.859,-43.792,178.616,5.998,149.485
C02412=1143.629,-114.610,-43.801,178.618,5.999,149.485
C02413=1143.624,-114.360,-43.810,178.619,5.999,149.484
C02414=1143.618,-114.111,-43.818,178.622,6.000,149.484
C02415=1143.613,-113.860,-43.827,178.623,6.000,149.483
C02416=1143.608,-113.610,-43.836,178.625,6.000,149.483
C02417=1143.602,-113.360,-43.844,178.627,6.000,149.482
C02418=1143.597,-113.111,-43.853,178.629,6.001,149.482
C02419=1143.591,-112.861,-43.862,178.631,6.001,149.481
C02420=1143.586,-112.612,-43.871,178.633,6.001,149.481
C02421=1143.581,-112.361,-43.879,178.636,6.002,149.480
C02422=1143.575,-112.112,-43.887,178.637,6.002,149.480
C02423=1143.570,-111.862,-43.896,178.639,6.003,149.479
C02424=1143.565,-111.612,-43.905,178.641,6.003,149.479
C02425=1143.559,-111.362,-43.914,178.643,6.004,149.478
C02426=1143.554,-111.113,-43.923,178.645,6.004,149.478
C02427=1143.549,-110.863,-43.932,178.647,6.004,149.477
C02428=1143.543,-110.614,-43.940,178.649,6.005,149.477
C02429=1143.538,-110.363,-43.949,178.651,6.005,149.476
C02430=1143.533,-110.113,-43.958,178.653,6.005,149.476
C02431=1143.527,-109.864,-43.966,178.655,6.005,149.475
C02432=1143.522,-109.614,-43.975,178.657,6.006,149.475
C02433=1143.516,-109.364,-43.984,178.659,6.007,149.474
C02434=1143.511,-109.114,-43.993,178.661,6.007,149.474
C02435=1143.506,-108.864,-44.002,178.663,6.008,149.473
C02436=1143.500,-108.614,-44.011,178.665,6.007,149.473
C02437=1143.495,-108.365,-44.020,178.668,6.008,149.472
C02438=1143.489,-108.115,-44.029,178.669,6.008,149.471
C02439=1143.484,-107.866,-44.038,178.671,6.009,149.471
C02440=1143.479,-107.616,-44.046,178.674,6.009,149.470
C02441=1143.474,-107.366,-44.055,178.675,6.009,149.470
C02442=1143.469,-107.116,-44.064,178.677,6.010,149.470
C02443=1143.462,-106.867,-44.073,178.679,6.010,149.469
C02444=1143.457,-106.617,-44.082,178.681,6.011,149.469
C02445=1143.452,-106.367,-44.091,178.684,6.011,149.468
C02446=1143.447,-106.117,-44.100,178.685,6.011,149.467
C02447=1143.442,-105.867,-44.109,178.688,6.012,149.467
C02448=1143.436,-105.617,-44.118,178.689,6.012,149.466
C02449=1143.430,-105.368,-44.127,178.691,6.013,149.466
C02450=1143.425,-105.118,-44.136,178.694,6.013,149.465
C02451=1143.420,-104.868,-44.145,178.695,6.013,149.465
C02452=1143.414,-104.618,-44.154,178.697,6.014,149.464
C02453=1143.409,-104.368,-44.163,178.699,6.014,149.464
C02454=1143.404,-104.119,-44.171,178.702,6.014,149.463
C02455=1143.398,-103.868,-44.181,178.704,6.015,149.463
C02456=1143.393,-103.619,-44.190,178.705,6.015,149.462
C02457=1143.387,-103.369,-44.198,178.708,6.016,149.462
C02458=1143.382,-103.098,-44.209,178.710,6.016,149.461
C02459=1143.376,-102.825,-44.218,178.712,6.016,149.461
C02460=1143.371,-102.553,-44.228,178.714,6.017,149.460
C02461=1143.365,-102.281,-44.238,178.717,6.017,149.459
C02462=1143.359,-102.031,-44.248,178.719,6.018,149.459
C02463=1143.354,-101.781,-44.257,178.721,6.018,149.458
C02464=1143.349,-101.531,-44.266,178.723,6.019,149.458
C02465=1143.344,-101.281,-44.275,178.724,6.019,149.457
C02466=1143.337,-101.032,-44.284,178.727,6.019,149.457
C02467=1143.332,-100.782,-44.293,178.729,6.020,149.456
C02468=1143.327,-100.532,-44.302,178.731,6.020,149.456
C02469=1143.322,-100.283,-44.311,178.733,6.020,149.455
C02470=1143.316,-100.033,-44.321,178.735,6.021,149.455
C02471=1143.311,-99.783,-44.330,178.737,6.021,149.454
C02472=1143.306,-99.533,-44.339,178.739,6.022,149.454
C02473=1143.301,-99.283,-44.347,178.741,6.022,149.453
C02474=1143.295,-99.034,-44.358,178.743,6.022,149.453
C02475=1143.290,-98.784,-44.367,178.745,6.023,149.452
C02476=1143.285,-98.534,-44.375,178.747,6.023,149.452
C02477=1143.279,-98.284,-44.385,178.749,6.024,149.451
C02478=1143.274,-98.034,-44.394,178.751,6.024,149.451
C02479=1143.269,-97.785,-44.403,178.753,6.024,149.450
C02480=1143.263,-97.535,-44.413,178.756,6.025,149.449
C02481=1143.257,-97.286,-44.422,178.758,6.026,149.449
C02482=1143.252,-97.036,-44.430,178.759,6.026,149.449
C02483=1143.246,-96.786,-44.441,178.762,6.026,149.448
C02484=1143.241,-96.536,-44.450,178.763,6.026,149.448
C02485=1143.236,-96.286,-44.458,178.766,6.027,149.447
C02486=1143.230,-96.036,-44.468,178.768,6.027,149.446
C02487=1143.225,-95.787,-44.478,178.770,6.027,149.446
C02488=1143.220,-95.537,-44.486,178.772,6.028,149.445
C02489=1143.214,-95.287,-44.496,178.774,6.029,149.445
C02490=1143.209,-95.038,-44.506,178.776,6.029,149.444
C02491=1143.204,-94.788,-44.514,178.778,6.029,149.444
C02492=1143.198,-94.538,-44.524,178.781,6.030,149.443
C02493=1143.193,-94.289,-44.534,178.782,6.030,149.443
C02494=1143.188,-94.039,-44.542,178.784,6.031,149.442
C02495=1143.182,-93.789,-44.552,178.787,6.031,149.442
C02496=1143.177,-93.539,-44.562,178.789,6.031,149.441
C02497=1143.171,-93.289,-44.571,178.791,6.032,149.441
C02498=1143.166,-93.039,-44.580,178.793,6.033,149.440
C02499=1143.161,-92.790,-44.590,178.795,6.032,149.440
C02500=1143.156,-92.540,-44.599,178.797,6.033,149.439
C02501=1143.150,-92.290,-44.608,178.800,6.034,149.438
C02502=1143.145,-92.040,-44.618,178.801,6.034,149.438
C02503=1143.140,-91.791,-44.627,178.803,6.034,149.437
C02504=1143.135,-91.540,-44.638,178.806,6.035,149.437
C02505=1143.129,-91.291,-44.647,178.807,6.035,149.436
C02506=1143.124,-91.041,-44.655,178.810,6.035,149.436
C02507=1143.119,-90.791,-44.666,178.812,6.036,149.435
C02508=1143.113,-90.541,-44.675,178.814,6.036,149.435
C02509=1143.108,-90.292,-44.685,178.816,6.037,149.434
C02510=1143.103,-90.042,-44.694,178.818,6.038,149.434
C02511=1143.097,-89.792,-44.704,178.820,6.037,149.433
C02512=1143.092,-89.543,-44.713,178.822,6.038,149.433
C02513=1143.086,-89.293,-44.723,178.824,6.039,149.432
C02514=1143.081,-89.043,-44.732,178.826,6.039,149.432
C02515=1143.076,-88.794,-44.742,178.828,6.039,149.431
C02516=1143.070,-88.544,-44.751,178.831,6.040,149.430
C02517=1143.065,-88.294,-44.760,178.832,6.040,149.430
C02518=1143.060,-88.044,-44.770,178.835,6.041,149.429
C02519=1143.054,-87.793,-44.780,178.837,6.041,149.429
C02520=1143.049,-87.544,-44.790,178.838,6.041,149.429
C02521=1143.044,-87.295,-44.800,178.841,6.042,149.428
C02522=1143.039,-87.045,-44.809,178.843,6.042,149.427
C02523=1143.033,-86.795,-44.819,178.846,6.043,149.427
C02524=1143.028,-86.545,-44.828,178.847,6.043,149.426
C02525=1143.022,-86.296,-44.838,178.850,6.044,149.426
C02526=1143.017,-86.046,-44.847,178.852,6.044,149.425
C02527=1143.012,-85.797,-44.857,178.854,6.044,149.425
C02528=1143.007,-85.546,-44.866,178.856,6.045,149.424
C02529=1143.001,-85.296,-44.877,178.858,6.046,149.424
C02530=1142.997,-85.047,-44.886,178.860,6.045,149.423
C02531=1142.991,-84.797,-44.896,178.862,6.046,149.423
C02532=1142.986,-84.548,-44.905,178.864,6.047,149.422
C02533=1142.980,-84.298,-44.915,178.867,6.048,149.422
C02534=1142.974,-84.048,-44.925,178.869,6.047,149.421
C02535=1142.969,-83.799,-44.935,178.871,6.048,149.420
C02536=1142.964,-83.548,-44.944,178.873,6.049,149.420
C02537=1142.959,-83.299,-44.954,178.875,6.049,149.419
C02538=1142.953,-83.049,-44.964,178.877,6.049,149.419
C02539=1142.949,-82.799,-44.973,178.880,6.050,149.418
C02540=1142.943,-82.550,-44.983,178.882,6.051,149.418
C02541=1142.937,-82.300,-44.993,178.883,6.051,149.417
C02542=1142.933,-82.050,-45.003,178.886,6.051,149.417
C02543=1142.927,-81.800,-45.013,178.888,6.052,149.416
C02544=1142.921,-81.550,-45.023,178.890,6.052,149.416
C02545=1142.916,-81.301,-45.032,178.892,6.052,149.415
C02546=1142.911,-81.051,-45.042,178.894,6.053,149.415
C02547=1142.906,-80.801,-45.051,178.897,6.054,149.414
C02548=1142.901,-80.551,-45.062,178.898,6.054,149.413
C02549=1142.895,-80.302,-45.072,178.901,6.054,149.413
C02550=1142.890,-80.052,-45.082,178.903,6.055,149.412
C02551=1142.884,-79.802,-45.091,178.905,6.055,149.412
C02552=1142.879,-79.553,-45.101,178.907,6.055,149.411
C02553=1142.874,-79.303,-45.111,178.909,6.056,149.411
C02554=1142.868,-79.053,-45.121,178.911,6.057,149.410
C02555=1142.863,-78.803,-45.131,178.914,6.057,149.410
C02556=1142.857,-78.553,-45.141,178.916,6.057,149.409
C02557=1142.852,-78.304,-45.151,178.918,6.058,149.409
C02558=1142.847,-78.053,-45.161,178.920,6.059,149.408
C02559=1142.842,-77.804,-45.171,178.922,6.058,149.407
C02560=1142.837,-77.555,-45.181,178.924,6.059,149.407
C02561=1142.831,-77.305,-45.191,178.927,6.060,149.406
C02562=1142.825,-77.033,-45.202,178.929,6.060,149.406
C02563=1142.820,-76.762,-45.212,178.931,6.061,149.405
C02564=1142.814,-76.491,-45.223,178.934,6.061,149.405
C02565=1142.808,-76.219,-45.235,178.936,6.061,149.404
C02566=1142.802,-75.969,-45.244,178.938,6.062,149.404
C02567=1142.798,-75.719,-45.254,178.941,6.063,149.403
C02568=1142.792,-75.470,-45.264,178.943,6.063,149.402
C02569=1142.787,-75.220,-45.274,178.944,6.063,149.402
C02570=1142.781,-74.971,-45.285,178.947,6.064,149.401
C02571=1142.777,-74.721,-45.295,178.949,6.064,149.401
C02572=1142.771,-74.471,-45.305,178.951,6.065,149.400
C02573=1142.765,-74.221,-45.314,178.953,6.065,149.400
C02574=1142.760,-73.971,-45.325,178.955,6.066,149.399
C02575=1142.755,-73.721,-45.335,178.958,6.066,149.399
C02576=1142.750,-73.472,-45.345,178.960,6.067,149.398
C02577=1142.744,-73.222,-45.355,178.962,6.067,149.398
C02578=1142.739,-72.972,-45.366,178.964,6.068,149.397
C02579=1142.734,-72.723,-45.376,178.967,6.068,149.396
C02580=1142.728,-72.473,-45.386,178.969,6.069,149.396
C02581=1142.723,-72.224,-45.396,178.971,6.070,149.395
C02582=1142.718,-71.974,-45.406,178.973,6.069,149.395
C02583=1142.713,-71.724,-45.416,178.975,6.070,149.394
C02584=1142.707,-71.475,-45.427,178.977,6.071,149.394
C02585=1142.702,-71.224,-45.436,178.980,6.072,149.393
C02586=1142.696,-70.974,-45.447,178.982,6.071,149.393
C02587=1142.690,-70.725,-45.457,178.984,6.072,149.392
C02588=1142.686,-70.475,-45.467,178.986,6.073,149.392
C02589=1142.681,-70.225,-45.477,178.989,6.073,149.391
C02590=1142.675,-69.976,-45.487,178.991,6.074,149.390
C02591=1142.670,-69.725,-45.498,178.992,6.074,149.390
C02592=1142.664,-69.476,-45.508,178.995,6.075,149.389
C02593=1142.659,-69.226,-45.518,178.997,6.075,149.389
C02594=1142.654,-68.976,-45.529,179.000,6.076,149.388
C02595=1142.648,-68.727,-45.540,179.001,6.076,149.388
C02596=1142.644,-68.478,-45.549,179.003,6.077,149.387
C02597=1142.639,-68.228,-45.560,179.006,6.077,149.387
C02598=1142.633,-67.978,-45.570,179.008,6.078,149.386
C02599=1142.627,-67.728,-45.580,179.010,6.078,149.386
C02600=1142.622,-67.478,-45.591,179.012,6.078,149.385
C02601=1142.617,-67.229,-45.601,179.015,6.079,149.384
C02602=1142.611,-66.979,-45.611,179.017,6.080,149.384
C02603=1142.606,-66.729,-45.622,179.020,6.080,149.383
C02604=1142.601,-66.479,-45.632,179.022,6.081,149.383
C02605=1142.596,-66.229,-45.643,179.023,6.081,149.382
C02606=1142.590,-65.980,-45.653,179.025,6.082,149.382
C02607=1142.585,-65.731,-45.664,179.028,6.082,149.381
C02608=1142.580,-65.480,-45.674,179.030,6.083,149.381
C02609=1142.575,-65.231,-45.684,179.033,6.083,149.380
C02610=1142.570,-64.981,-45.695,179.035,6.083,149.379
C02611=1142.564,-64.731,-45.705,179.037,6.084,149.379
C02612=1142.559,-64.482,-45.715,179.039,6.085,149.378
C02613=1142.554,-64.232,-45.726,179.041,6.085,149.378
C02614=1142.548,-63.983,-45.737,179.044,6.086,149.377
C02615=1142.543,-63.732,-45.747,179.045,6.086,149.377
C02616=1142.538,-63.483,-45.757,179.048,6.086,149.376
C02617=1142.533,-63.233,-45.768,179.050,6.087,149.376
C02618=1142.527,-62.983,-45.778,179.052,6.088,149.375
C02619=1142.522,-62.734,-45.789,179.055,6.088,149.375
C02620=1142.517,-62.484,-45.800,179.057,6.089,149.374
C02621=1142.511,-62.234,-45.810,179.059,6.089,149.373
C02622=1142.506,-61.984,-45.820,179.061,6.090,149.373
C02623=1142.501,-61.735,-45.831,179.064,6.090,149.372
C02624=1142.496,-61.485,-45.842,179.066,6.091,149.372
C02625=1142.490,-61.235,-45.853,179.068,6.091,149.371
C02626=1142.485,-60.985,-45.863,179.070,6.091,149.371
C02627=1142.479,-60.736,-45.874,179.072,6.092,149.370
C02628=1142.474,-60.486,-45.885,179.075,6.093,149.370
C02629=1142.469,-60.236,-45.895,179.077,6.093,149.369
C02630=1142.464,-59.986,-45.906,179.079,6.094,149.368
C02631=1142.459,-59.737,-45.916,179.082,6.095,149.368
C02632=1142.453,-59.487,-45.927,179.083,6.095,149.368
C02633=1142.448,-59.237,-45.937,179.086,6.095,149.367
C02634=1142.443,-58.988,-45.948,179.088,6.096,149.366
C02635=1142.438,-58.738,-45.959,179.090,6.096,149.366
C02636=1142.432,-58.488,-45.969,179.093,6.097,149.365
C02637=1142.427,-58.239,-45.980,179.095,6.098,149.365
C02638=1142.422,-57.989,-45.990,179.097,6.098,149.364
C02639=1142.416,-57.739,-46.002,179.099,6.098,149.363
C02640=1142.411,-57.489,-46.013,179.102,6.099,149.363
C02641=1142.406,-57.240,-46.023,179.104,6.100,149.363
C02642=1142.401,-56.990,-46.034,179.106,6.100,149.362
C02643=1142.395,-56.740,-46.045,179.109,6.101,149.361
C02644=1142.390,-56.490,-46.055,179.111,6.101,149.361
C02645=1142.385,-56.241,-46.066,179.112,6.101,149.360
C02646=1142.380,-55.991,-46.077,179.115,6.102,149.360
C02647=1142.374,-55.742,-46.088,179.117,6.103,149.359
C02648=1142.369,-55.492,-46.099,179.119,6.103,149.359
C02649=1142.364,-55.242,-46.109,179.122,6.104,149.358
C02650=1142.359,-54.992,-46.120,179.124,6.105,149.358
C02651=1142.353,-54.743,-46.130,179.127,6.105,149.357
C02652=1142.349,-54.493,-46.142,179.129,6.106,149.356
C02653=1142.343,-54.243,-46.153,179.131,6.106,149.356
C02654=1142.338,-53.994,-46.164,179.133,6.106,149.355
C02655=1142.333,-53.743,-46.174,179.136,6.107,149.355
C02656=1142.327,-53.495,-46.185,179.138,6.108,149.354
C02657=1142.322,-53.244,-46.196,179.140,6.108,149.354
C02658=1142.316,-52.995,-46.207,179.143,6.109,149.353
C02659=1142.311,-52.745,-46.218,179.145,6.110,149.353
C02660=1142.307,-52.495,-46.229,179.146,6.110,149.352
C02661=1142.301,-52.246,-46.240,179.149,6.110,149.351
C02662=1142.295,-51.996,-46.251,179.151,6.111,149.351
C02663=1142.290,-51.746,-46.262,179.154,6.112,149.350
C02664=1142.285,-51.497,-46.273,179.156,6.112,149.350
C02665=1142.280,-51.246,-46.283,179.158,6.113,149.349
C02666=1142.274,-50.976,-46.295,179.161,6.113,149.349
C02667=1142.268,-50.705,-46.308,179.163,6.114,149.348
C02668=1142.262,-50.435,-46.319,179.166,6.114,149.347
C02669=1142.257,-50.164,-46.331,179.168,6.115,149.347
C02670=1142.252,-49.914,-46.343,179.170,6.116,149.346
C02671=1142.246,-49.665,-46.353,179.173,6.116,149.346
C02672=1142.242,-49.415,-46.365,179.175,6.117,149.345
C02673=1142.236,-49.164,-46.376,179.178,6.117,149.344
C02674=1142.231,-48.916,-46.387,179.180,6.118,149.344
C02675=1142.226,-48.666,-46.398,179.182,6.118,149.344
C02676=1142.220,-48.415,-46.409,179.184,6.119,149.343
C02677=1142.215,-48.166,-46.420,179.186,6.119,149.342
C02678=1142.210,-47.917,-46.431,179.189,6.120,149.342
C02679=1142.204,-47.667,-46.442,179.191,6.120,149.341
C02680=1142.199,-47.417,-46.453,179.194,6.121,149.341
C02681=1142.194,-47.168,-46.465,179.196,6.122,149.340
C02682=1142.188,-46.918,-46.475,179.198,6.122,149.340
C02683=1142.183,-46.668,-46.487,179.201,6.123,149.339
C02684=1142.179,-46.419,-46.498,179.203,6.124,149.339
C02685=1142.172,-46.169,-46.509,179.205,6.124,149.338
C02686=1142.168,-45.919,-46.520,179.207,6.124,149.337
C02687=1142.162,-45.669,-46.532,179.209,6.125,149.337
C02688=1142.158,-45.420,-46.543,179.212,6.126,149.336
C02689=1142.152,-45.170,-46.554,179.214,6.126,149.336
C02690=1142.146,-44.920,-46.565,179.216,6.127,149.335
C02691=1142.142,-44.670,-46.577,179.219,6.127,149.335
C02692=1142.136,-44.421,-46.588,179.221,6.128,149.334
C02693=1142.131,-44.171,-46.599,179.223,6.129,149.334
C02694=1142.126,-43.921,-46.610,179.226,6.129,149.333
C02695=1142.120,-43.672,-46.622,179.228,6.130,149.332
C02696=1142.115,-43.422,-46.633,179.230,6.131,149.332
C02697=1142.110,-43.173,-46.645,179.233,6.131,149.331
C02698=1142.105,-42.922,-46.655,179.235,6.131,149.331
C02699=1142.099,-42.673,-46.667,179.237,6.132,149.330
C02700=1142.094,-42.423,-46.678,179.239,6.133,149.330
C02701=1142.090,-42.174,-46.689,179.242,6.133,149.329
C02702=1142.084,-41.924,-46.701,179.244,6.134,149.328
C02703=1142.079,-41.675,-46.712,179.246,6.135,149.328
C02704=1142.073,-41.424,-46.723,179.249,6.135,149.327
C02705=1142.068,-41.175,-46.735,179.251,6.136,149.327
C02706=1142.063,-40.925,-46.747,179.253,6.137,149.326
C02707=1142.058,-40.676,-46.758,179.256,6.137,149.326
C02708=1142.052,-40.426,-46.769,179.258,6.138,149.325
C02709=1142.048,-40.176,-46.781,179.261,6.138,149.325
C02710=1142.042,-39.926,-46.793,179.263,6.139,149.324
C02711=1142.037,-39.677,-46.804,179.265,6.140,149.323
C02712=1142.031,-39.427,-46.815,179.268,6.140,149.323
C02713=1142.026,-39.177,-46.826,179.270,6.141,149.322
C02714=1142.021,-38.927,-46.838,179.272,6.142,149.322
C02715=1142.016,-38.678,-46.849,179.275,6.142,149.321
C02716=1142.010,-38.428,-46.861,179.277,6.142,149.321
C02717=1142.005,-38.179,-46.873,179.279,6.143,149.320
C02718=1142.000,-37.929,-46.884,179.281,6.144,149.320
C02719=1141.995,-37.679,-46.896,179.284,6.144,149.319
C02720=1141.989,-37.430,-46.907,179.286,6.145,149.318
C02721=1141.984,-37.180,-46.919,179.288,6.146,149.318
C02722=1141.979,-36.930,-46.930,179.291,6.146,149.317
C02723=1141.974,-36.681,-46.942,179.293,6.147,149.317
C02724=1141.968,-36.431,-46.954,179.296,6.147,149.316
C02725=1141.963,-36.182,-46.965,179.298,6.148,149.316
C02726=1141.958,-35.932,-46.976,179.300,6.149,149.315
C02727=1141.953,-35.682,-46.988,179.303,6.149,149.314
C02728=1141.948,-35.432,-47.000,179.305,6.150,149.314
C02729=1141.942,-35.182,-47.011,179.307,6.151,149.314
C02730=1141.937,-34.933,-47.023,179.310,6.151,149.313
C02731=1141.931,-34.683,-47.034,179.312,6.152,149.312
C02732=1141.927,-34.434,-47.046,179.314,6.153,149.312
C02733=1141.921,-34.184,-47.057,179.317,6.153,149.311
C02734=1141.916,-33.935,-47.070,179.319,6.154,149.311
C02735=1141.911,-33.685,-47.081,179.322,6.154,149.310
C02736=1141.906,-33.435,-47.093,179.324,6.155,149.310
C02737=1141.901,-33.185,-47.105,179.326,6.156,149.309
C02738=1141.896,-32.935,-47.116,179.329,6.156,149.308
C02739=1141.890,-32.686,-47.128,179.331,6.157,149.308
C02740=1141.884,-32.436,-47.140,179.333,6.158,149.307
C02741=1141.880,-32.187,-47.151,179.336,6.158,149.307
C02742=1141.875,-31.937,-47.164,179.338,6.159,149.306
C02743=1141.869,-31.687,-47.176,179.340,6.159,149.306
C02744=1141.865,-31.438,-47.187,179.343,6.160,149.305
C02745=1141.859,-31.188,-47.199,179.345,6.161,149.305
C02746=1141.854,-30.938,-47.211,179.348,6.161,149.304
C02747=1141.848,-30.688,-47.223,179.350,6.162,149.303
C02748=1141.844,-30.439,-47.235,179.352,6.163,149.303
C02749=1141.838,-30.190,-47.246,179.355,6.163,149.302
C02750=1141.832,-29.940,-47.258,179.357,6.164,149.302
C02751=1141.827,-29.690,-47.270,179.359,6.165,149.301
C02752=1141.822,-29.440,-47.281,179.362,6.165,149.301
C02753=1141.817,-29.191,-47.294,179.364,6.166,149.300
C02754=1141.812,-28.941,-47.306,179.366,6.167,149.299
C02755=1141.807,-28.691,-47.317,179.369,6.167,149.299
C02756=1141.802,-28.441,-47.329,179.371,6.168,149.298
C02757=1141.796,-28.192,-47.341,179.373,6.169,149.298
C02758=1141.791,-27.942,-47.353,179.376,6.169,149.297
C02759=1141.786,-27.692,-47.365,179.378,6.170,149.297
C02760=1141.781,-27.443,-47.377,179.380,6.171,149.296
C02761=1141.776,-27.193,-47.389,179.383,6.171,149.296
C02762=1141.770,-26.943,-47.401,179.385,6.172,149.295
C02763=1141.765,-26.694,-47.414,179.388,6.173,149.295
C02764=1141.760,-26.444,-47.425,179.390,6.173,149.294
C02765=1141.755,-26.194,-47.437,179.392,6.174,149.293
C02766=1141.750,-25.945,-47.449,179.395,6.175,149.293
C02767=1141.745,-25.695,-47.461,179.397,6.175,149.292
C02768=1141.739,-25.445,-47.473,179.399,6.176,149.292
C02769=1141.734,-25.196,-47.486,179.402,6.177,149.291
C02770=1141.728,-24.926,-47.498,179.405,6.178,149.291
C02771=1141.723,-24.656,-47.511,179.407,6.179,149.290
C02772=1141.717,-24.386,-47.524,179.410,6.179,149.289
C02773=1141.712,-24.116,-47.537,179.412,6.179,149.289
C02774=1141.706,-23.867,-47.549,179.415,6.180,149.288
C02775=1141.701,-23.617,-47.561,179.417,6.181,149.288
C02776=1141.696,-23.367,-47.574,179.419,6.181,149.287
C02777=1141.690,-23.117,-47.586,179.422,6.182,149.287
C02778=1141.685,-22.867,-47.598,179.424,6.183,149.286
C02779=1141.680,-22.618,-47.610,179.426,6.183,149.285
C02780=1141.674,-22.368,-47.622,179.429,6.185,149.285
C02781=1141.669,-22.119,-47.635,179.432,6.185,149.284
C02782=1141.664,-21.869,-47.647,179.434,6.186,149.284
C02783=1141.660,-21.620,-47.659,179.436,6.187,149.283
C02784=1141.654,-21.370,-47.671,179.439,6.187,149.283
C02785=1141.650,-21.120,-47.684,179.441,6.188,149.282
C02786=1141.644,-20.870,-47.695,179.444,6.189,149.281
C02787=1141.639,-20.621,-47.708,179.446,6.189,149.281
C02788=1141.634,-20.371,-47.720,179.448,6.190,149.280
C02789=1141.628,-20.121,-47.732,179.451,6.191,149.280
C02790=1141.623,-19.872,-47.744,179.453,6.191,149.279
C02791=1141.618,-19.622,-47.757,179.456,6.192,149.279
C02792=1141.613,-19.373,-47.770,179.458,6.193,149.278
C02793=1141.607,-19.123,-47.781,179.460,6.193,149.278
C02794=1141.602,-18.874,-47.794,179.463,6.194,149.277
C02795=1141.597,-18.624,-47.806,179.465,6.195,149.276
C02796=1141.592,-18.374,-47.819,179.468,6.196,149.276
C02797=1141.586,-18.124,-47.830,179.470,6.197,149.275
C02798=1141.582,-17.874,-47.843,179.472,6.197,149.275
C02799=1141.577,-17.625,-47.856,179.475,6.198,149.274
C02800=1141.571,-17.375,-47.868,179.477,6.199,149.274
C02801=1141.566,-17.126,-47.880,179.479,6.199,149.273
C02802=1141.561,-16.877,-47.893,179.482,6.200,149.273
C02803=1141.556,-16.627,-47.905,179.484,6.201,149.272
C02804=1141.550,-16.377,-47.918,179.487,6.201,149.271
C02805=1141.545,-16.127,-47.929,179.489,6.202,149.271
C02806=1141.540,-15.877,-47.942,179.491,6.203,149.270
C02807=1141.535,-15.628,-47.955,179.495,6.204,149.270
C02808=1141.530,-15.379,-47.968,179.497,6.205,149.269
C02809=1141.524,-15.128,-47.980,179.499,6.205,149.269
C02810=1141.519,-14.879,-47.993,179.502,6.206,149.268
C02811=1141.514,-14.630,-48.005,179.504,6.207,149.268
C02812=1141.509,-14.379,-48.018,179.506,6.207,149.267
C02813=1141.504,-14.130,-48.030,179.509,6.208,149.266
C02814=1141.499,-13.881,-48.043,179.511,6.208,149.266
C02815=1141.494,-13.631,-48.055,179.513,6.209,149.265
C02816=1141.488,-13.381,-48.067,179.516,6.210,149.265
C02817=1141.483,-13.132,-48.080,179.519,6.211,149.264
C02818=1141.478,-12.882,-48.093,179.521,6.212,149.264
C02819=1141.473,-12.632,-48.106,179.523,6.213,149.263
C02820=1141.467,-12.382,-48.118,179.526,6.213,149.263
C02821=1141.462,-12.133,-48.130,179.528,6.214,149.262
C02822=1141.457,-11.884,-48.143,179.531,6.214,149.261
C02823=1141.452,-11.634,-48.156,179.533,6.215,149.261
C02824=1141.447,-11.384,-48.169,179.535,6.216,149.260
C02825=1141.442,-11.135,-48.181,179.538,6.217,149.260
C02826=1141.436,-10.885,-48.194,179.541,6.218,149.259
C02827=1141.431,-10.635,-48.207,179.543,6.218,149.259
C02828=1141.426,-10.386,-48.219,179.545,6.219,149.258
C02829=1141.421,-10.136,-48.232,179.548,6.220,149.258
C02830=1141.416,-9.887,-48.245,179.550,6.220,149.257
C02831=1141.410,-9.637,-48.258,179.552,6.221,149.256
C02832=1141.406,-9.387,-48.271,179.555,6.222,149.256
C02833=1141.401,-9.138,-48.283,179.558,6.223,149.255
C02834=1141.395,-8.888,-48.295,179.560,6.224,149.255
C02835=1141.390,-8.639,-48.308,179.563,6.224,149.254
C02836=1141.385,-8.388,-48.321,179.565,6.225,149.254
C02837=1141.380,-8.139,-48.334,179.567,6.226,149.253
C02838=1141.375,-7.890,-48.347,179.570,6.226,149.253
C02839=1141.370,-7.640,-48.359,179.572,6.227,149.252
C02840=1141.364,-7.390,-48.373,179.575,6.228,149.251
C02841=1141.359,-7.141,-48.385,179.577,6.229,149.251
C02842=1141.354,-6.891,-48.398,179.580,6.230,149.250
C02843=1141.349,-6.641,-48.411,179.582,6.230,149.250
C02844=1141.344,-6.392,-48.424,179.584,6.231,149.249
C02845=1141.338,-6.142,-48.437,179.587,6.232,149.249
C02846=1141.334,-5.892,-48.450,179.590,6.233,149.248
C02847=1141.328,-5.643,-48.463,179.592,6.234,149.248
C02848=1141.323,-5.393,-48.475,179.595,6.234,149.247
C02849=1141.318,-5.144,-48.488,179.597,6.235,149.246
C02850=1141.313,-4.894,-48.502,179.599,6.236,149.246
C02851=1141.307,-4.645,-48.514,179.602,6.237,149.245
C02852=1141.302,-4.395,-48.527,179.604,6.237,149.245
C02853=1141.297,-4.145,-48.540,179.607,6.239,149.244
C02854=1141.292,-3.896,-48.553,179.609,6.239,149.244
C02855=1141.287,-3.646,-48.566,179.612,6.240,149.243
C02856=1141.282,-3.397,-48.580,179.614,6.241,149.243
C02857=1141.277,-3.147,-48.592,179.616,6.241,149.242
C02858=1141.272,-2.898,-48.605,179.619,6.243,149.241
C02859=1141.266,-2.648,-48.619,179.622,6.243,149.241
C02860=1141.261,-2.398,-48.631,179.624,6.244,149.240
C02861=1141.257,-2.148,-48.644,179.626,6.245,149.240
C02862=1141.251,-1.899,-48.657,179.629,6.245,149.239
C02863=1141.246,-1.649,-48.670,179.631,6.246,149.239
C02864=1141.241,-1.400,-48.684,179.634,6.247,149.238
C02865=1141.236,-1.150,-48.697,179.637,6.248,149.237
C02866=1141.230,-0.901,-48.709,179.639,6.249,149.237
C02867=1141.225,-0.651,-48.723,179.641,6.250,149.237
C02868=1141.220,-0.401,-48.736,179.644,6.250,149.236
C02869=1141.215,-0.151,-48.749,179.647,6.252,149.235
C02870=1141.210,0.098,-48.762,179.649,6.252,149.235
C02871=1141.204,0.347,-48.776,179.651,6.253,149.234
C02872=1141.200,0.597,-48.789,179.654,6.254,149.234
C02873=1141.194,0.847,-48.802,179.656,6.254,149.233
C02874=1141.189,1.116,-48.816,179.659,6.256,149.233
C02875=1141.183,1.386,-48.830,179.662,6.256,149.232
C02876=1141.177,1.655,-48.845,179.665,6.257,149.231
C02877=1141.172,1.925,-48.859,179.667,6.258,149.231
C02878=1141.166,2.174,-48.872,179.669,6.259,149.230
C02879=1141.162,2.424,-48.886,179.672,6.259,149.230
C02880=1141.156,2.673,-48.899,179.675,6.261,149.229
C02881=1141.152,2.923,-48.912,179.677,6.261,149.228
C02882=1141.146,3.172,-48.926,179.680,6.262,149.228
C02883=1141.142,3.422,-48.939,179.682,6.263,149.228
C02884=1141.136,3.672,-48.952,179.684,6.263,149.227
C02885=1141.132,3.921,-48.966,179.687,6.265,149.226
C02886=1141.126,4.171,-48.979,179.690,6.265,149.226
C02887=1141.121,4.420,-48.991,179.692,6.266,149.225
C02888=1141.116,4.670,-49.006,179.694,6.267,149.225
C02889=1141.110,4.920,-49.019,179.697,6.268,149.224
C02890=1141.105,5.170,-49.032,179.700,6.269,149.224
C02891=1141.100,5.419,-49.046,179.702,6.270,149.223
C02892=1141.095,5.669,-49.059,179.704,6.270,149.222
C02893=1141.090,5.918,-49.073,179.707,6.271,149.222
C02894=1141.085,6.168,-49.086,179.710,6.272,149.221
C02895=1141.080,6.417,-49.099,179.712,6.273,149.221
C02896=1141.074,6.667,-49.113,179.715,6.274,149.220
C02897=1141.069,6.916,-49.126,179.717,6.274,149.220
C02898=1141.064,7.166,-49.140,179.720,6.276,149.219
C02899=1141.059,7.415,-49.153,179.722,6.276,149.219
C02900=1141.054,7.665,-49.167,179.724,6.277,149.218
C02901=1141.048,7.915,-49.180,179.727,6.278,149.217
C02902=1141.044,8.164,-49.194,179.730,6.279,149.217
C02903=1141.039,8.414,-49.207,179.732,6.280,149.216
C02904=1141.033,8.663,-49.221,179.735,6.281,149.216
C02905=1141.029,8.913,-49.234,179.737,6.281,149.215
C02906=1141.023,9.162,-49.248,179.740,6.283,149.215
C02907=1141.018,9.413,-49.262,179.742,6.283,149.214
C02908=1141.013,9.662,-49.275,179.744,6.284,149.214
C02909=1141.008,9.911,-49.289,179.747,6.285,149.213
C02910=1141.002,10.161,-49.302,179.750,6.286,149.213
C02911=1140.998,10.410,-49.316,179.752,6.287,149.212
C02912=1140.993,10.661,-49.330,179.755,6.288,149.211
C02913=1140.987,10.910,-49.344,179.757,6.288,149.211
C02914=1140.983,11.160,-49.357,179.760,6.290,149.210
C02915=1140.977,11.409,-49.370,179.762,6.290,149.210
C02916=1140.972,11.658,-49.385,179.764,6.291,149.209
C02917=1140.966,11.908,-49.398,179.768,6.292,149.209
C02918=1140.962,12.157,-49.412,179.770,6.293,149.208
C02919=1140.957,12.407,-49.426,179.773,6.294,149.208
C02920=1140.951,12.657,-49.439,179.775,6.295,149.207
C02921=1140.946,12.906,-49.453,179.777,6.296,149.207
C02922=1140.942,13.155,-49.467,179.780,6.297,149.206
C02923=1140.936,13.405,-49.480,179.782,6.297,149.205
C02924=1140.931,13.655,-49.494,179.786,6.299,149.205
C02925=1140.926,13.904,-49.508,179.788,6.299,149.204
C02926=1140.921,14.154,-49.521,179.790,6.300,149.204
C02927=1140.916,14.404,-49.536,179.793,6.301,149.203
C02928=1140.911,14.653,-49.550,179.795,6.302,149.203
C02929=1140.906,14.903,-49.564,179.797,6.303,149.202
C02930=1140.901,15.153,-49.577,179.800,6.304,149.202
C02931=1140.896,15.402,-49.591,179.803,6.305,149.201
C02932=1140.891,15.651,-49.605,179.806,6.306,149.200
C02933=1140.885,15.900,-49.619,179.808,6.306,149.200
C02934=1140.880,16.151,-49.632,179.810,6.307,149.200
C02935=1140.875,16.400,-49.647,179.813,6.308,149.199
C02936=1140.869,16.649,-49.661,179.815,6.309,149.198
C02937=1140.865,16.899,-49.675,179.818,6.310,149.198
C02938=1140.860,17.149,-49.689,179.821,6.311,149.197
C02939=1140.855,17.399,-49.702,179.823,6.312,149.197
C02940=1140.850,17.648,-49.716,179.826,6.313,149.196
C02941=1140.845,17.898,-49.730,179.828,6.314,149.196
C02942=1140.840,18.147,-49.745,179.831,6.315,149.195
C02943=1140.834,18.396,-49.759,179.833,6.315,149.194
C02944=1140.829,18.646,-49.773,179.836,6.317,149.194
C02945=1140.824,18.896,-49.786,179.839,6.318,149.193
C02946=1140.818,19.145,-49.800,179.841,6.318,149.193
C02947=1140.814,19.395,-49.814,179.844,6.320,149.192
C02948=1140.809,19.644,-49.828,179.846,6.320,149.192
C02949=1140.804,19.894,-49.843,179.848,6.321,149.191
C02950=1140.799,20.143,-49.856,179.852,6.322,149.191
C02951=1140.794,20.393,-49.871,179.854,6.323,149.190
C02952=1140.789,20.643,-49.885,179.856,6.324,149.190
C02953=1140.784,20.892,-49.899,179.859,6.325,149.189
C02954=1140.778,21.141,-49.913,179.861,6.326,149.189
C02955=1140.773,21.391,-49.927,179.864,6.327,149.188
C02956=1140.768,21.641,-49.942,179.867,6.328,149.187
C02957=1140.763,21.890,-49.956,179.869,6.329,149.187
C02958=1140.758,22.139,-49.970,179.872,6.329,149.186
C02959=1140.753,22.389,-49.984,179.874,6.331,149.186
C02960=1140.748,22.639,-49.998,179.877,6.332,149.185
C02961=1140.743,22.889,-50.013,179.879,6.332,149.185
C02962=1140.737,23.138,-50.027,179.882,6.334,149.184
C02963=1140.732,23.387,-50.041,179.885,6.334,149.184
C02964=1140.727,23.637,-50.055,179.887,6.335,149.183
C02965=1140.722,23.887,-50.069,179.890,6.337,149.183
C02966=1140.718,24.136,-50.084,179.892,6.337,149.182
C02967=1140.712,24.385,-50.098,179.894,6.338,149.182
C02968=1140.707,24.635,-50.112,179.897,6.340,149.181
C02969=1140.702,24.885,-50.126,179.900,6.340,149.180
C02970=1140.697,25.135,-50.141,179.902,6.341,149.180
C02971=1140.692,25.384,-50.155,179.905,6.342,149.179
C02972=1140.687,25.633,-50.170,179.907,6.343,149.179
C02973=1140.681,25.883,-50.184,179.910,6.345,149.178
C02974=1140.676,26.132,-50.199,179.913,6.345,149.178
C02975=1140.671,26.382,-50.213,179.915,6.346,149.177
C02976=1140.666,26.632,-50.227,179.918,6.348,149.177
C02977=1140.661,26.882,-50.241,179.920,6.348,149.176
C02978=1140.656,27.150,-50.257,179.923,6.350,149.176
C02979=1140.651,27.418,-50.272,179.926,6.350,149.175
C02980=1140.644,27.688,-50.288,179.929,6.351,149.174
C02981=1140.639,27.957,-50.304,179.931,6.352,149.174
C02982=1140.634,28.207,-50.318,179.934,6.354,149.173
C02983=1140.629,28.456,-50.332,179.937,6.354,149.173
C02984=1140.625,28.705,-50.347,179.939,6.355,149.172
C02985=1140.619,28.955,-50.362,179.942,6.356,149.172
C02986=1140.614,29.205,-50.376,179.944,6.357,149.171
C02987=1140.608,29.454,-50.390,179.947,6.359,149.171
C02988=1140.604,29.703,-50.405,179.950,6.359,149.170
C02989=1140.599,29.953,-50.420,179.952,6.360,149.169
C02990=1140.594,30.203,-50.434,179.954,6.362,149.169
C02991=1140.589,30.452,-50.449,179.957,6.362,149.168
C02992=1140.584,30.702,-50.464,179.960,6.364,149.168
C02993=1140.579,30.952,-50.478,179.963,6.364,149.167
C02994=1140.574,31.201,-50.493,179.965,6.365,149.167
C02995=1140.569,31.450,-50.507,179.967,6.367,149.166
C02996=1140.563,31.700,-50.522,179.970,6.367,149.166
C02997=1140.559,31.949,-50.537,179.973,6.369,149.165
C02998=1140.554,32.199,-50.551,179.975,6.370,149.165
C02999=1140.549,32.449,-50.566,179.978,6.370,149.164
C03000=1140.543,32.698,-50.581,179.980,6.372,149.164
C03001=1140.538,32.947,-50.595,179.983,6.372,149.163
C03002=1140.533,33.196,-50.610,179.986,6.374,149.162
C03003=1140.527,33.446,-50.625,179.988,6.375,149.162
C03004=1140.523,33.696,-50.639,179.991,6.376,149.161
C03005=1140.518,33.945,-50.654,179.993,6.377,149.161
C03006=1140.513,34.195,-50.669,179.996,6.377,149.160
C03007=1140.508,34.444,-50.684,179.999,6.379,149.160
C03008=1140.503,34.694,-50.699,-179.999,6.380,149.159
C03009=1140.498,34.943,-50.713,-179.996,6.381,149.159
C03010=1140.492,35.193,-50.728,-179.994,6.382,149.158
C03011=1140.488,35.442,-50.743,-179.991,6.383,149.158
C03012=1140.483,35.692,-50.758,-179.989,6.384,149.157
C03013=1140.477,35.941,-50.773,-179.986,6.385,149.157
C03014=1140.472,36.191,-50.788,-179.983,6.386,149.156
C03015=1140.468,36.440,-50.802,-179.981,6.387,149.155
C03016=1140.462,36.690,-50.817,-179.978,6.388,149.155
C03017=1140.457,36.939,-50.832,-179.976,6.389,149.155
C03018=1140.452,37.189,-50.847,-179.972,6.390,149.154
C03019=1140.447,37.438,-50.862,-179.970,6.391,149.153
C03020=1140.442,37.688,-50.877,-179.967,6.393,149.153
C03021=1140.437,37.937,-50.892,-179.965,6.393,149.152
C03022=1140.432,38.187,-50.907,-179.963,6.394,149.152
C03023=1140.426,38.437,-50.922,-179.960,6.396,149.151
C03024=1140.422,38.686,-50.937,-179.957,6.396,149.151
C03025=1140.416,38.936,-50.952,-179.955,6.398,149.150
C03026=1140.412,39.185,-50.967,-179.952,6.399,149.150
C03027=1140.407,39.435,-50.982,-179.949,6.400,149.149
C03028=1140.402,39.685,-50.997,-179.947,6.401,149.149
C03029=1140.397,39.934,-51.012,-179.944,6.402,149.148
C03030=1140.391,40.183,-51.028,-179.942,6.403,149.148
C03031=1140.387,40.433,-51.042,-179.939,6.404,149.147
C03032=1140.381,40.682,-51.057,-179.936,6.405,149.147
C03033=1140.376,40.931,-51.072,-179.933,6.407,149.146
C03034=1140.371,41.181,-51.087,-179.931,6.407,149.146
C03035=1140.366,41.430,-51.102,-179.928,6.409,149.145
C03036=1140.361,41.680,-51.118,-179.926,6.409,149.144
C03037=1140.356,41.929,-51.133,-179.923,6.411,149.144
C03038=1140.351,42.180,-51.148,-179.920,6.412,149.143
C03039=1140.346,42.429,-51.163,-179.918,6.412,149.143
C03040=1140.341,42.678,-51.179,-179.915,6.414,149.142
C03041=1140.336,42.927,-51.194,-179.913,6.414,149.142
C03042=1140.331,43.177,-51.209,-179.910,6.416,149.141
C03043=1140.326,43.426,-51.224,-179.908,6.417,149.141
C03044=1140.321,43.676,-51.239,-179.905,6.418,149.140
C03045=1140.316,43.925,-51.254,-179.903,6.419,149.140
C03046=1140.311,44.175,-51.270,-179.900,6.421,149.139
C03047=1140.305,44.425,-51.285,-179.897,6.421,149.139
C03048=1140.301,44.674,-51.300,-179.894,6.423,149.138
C03049=1140.295,44.923,-51.316,-179.892,6.423,149.138
C03050=1140.291,45.173,-51.331,-179.889,6.425,149.137
C03051=1140.285,45.422,-51.346,-179.887,6.426,149.137
C03052=1140.281,45.672,-51.362,-179.884,6.427,149.136
C03053=1140.276,45.921,-51.377,-179.881,6.428,149.136
C03054=1140.270,46.171,-51.392,-179.879,6.429,149.135
C03055=1140.266,46.420,-51.407,-179.876,6.430,149.134
C03056=1140.260,46.670,-51.423,-179.873,6.432,149.134
C03057=1140.255,46.920,-51.439,-179.871,6.432,149.134
C03058=1140.251,47.169,-51.454,-179.868,6.434,149.133
C03059=1140.245,47.418,-51.469,-179.865,6.435,149.132
C03060=1140.240,47.668,-51.485,-179.863,6.436,149.132
C03061=1140.235,47.917,-51.500,-179.860,6.437,149.131
C03062=1140.231,48.167,-51.516,-179.858,6.438,149.131
C03063=1140.225,48.416,-51.531,-179.855,6.440,149.130
C03064=1140.221,48.665,-51.546,-179.852,6.440,149.130
C03065=1140.215,48.915,-51.562,-179.849,6.442,149.129
C03066=1140.210,49.165,-51.578,-179.847,6.443,149.129
C03067=1140.206,49.414,-51.593,-179.844,6.444,149.128
C03068=1140.200,49.663,-51.608,-179.842,6.445,149.128
C03069=1140.195,49.913,-51.624,-179.839,6.447,149.127
C03070=1140.191,50.163,-51.639,-179.836,6.447,149.127
C03071=1140.186,50.412,-51.655,-179.834,6.449,149.126
C03072=1140.180,50.661,-51.670,-179.831,6.449,149.126
C03073=1140.175,50.911,-51.686,-179.828,6.451,149.125
C03074=1140.171,51.161,-51.701,-179.826,6.452,149.125
C03075=1140.166,51.409,-51.718,-179.823,6.453,149.124
C03076=1140.160,51.659,-51.733,-179.820,6.454,149.124
C03077=1140.155,51.909,-51.749,-179.818,6.455,149.123
C03078=1140.151,52.158,-51.764,-179.815,6.457,149.123
C03079=1140.145,52.407,-51.780,-179.813,6.457,149.122
C03080=1140.140,52.657,-51.795,-179.810,6.459,149.122
C03081=1140.135,52.907,-51.811,-179.808,6.460,149.121
C03082=1140.130,53.175,-51.828,-179.804,6.461,149.120
C03083=1140.124,53.444,-51.845,-179.802,6.463,149.120
C03084=1140.119,53.712,-51.862,-179.798,6.464,149.119
C03085=1140.114,53.980,-51.879,-179.796,6.465,149.119
C03086=1140.109,54.231,-51.895,-179.793,6.467,149.118
C03087=1140.104,54.480,-51.910,-179.790,6.468,149.118
C03088=1140.099,54.729,-51.927,-179.788,6.469,149.117
C03089=1140.094,54.979,-51.943,-179.785,6.470,149.117
C03090=1140.088,55.228,-51.958,-179.783,6.471,149.116
C03091=1140.083,55.478,-51.974,-179.780,6.472,149.116
C03092=1140.079,55.727,-51.990,-179.778,6.473,149.115
C03093=1140.074,55.976,-52.005,-179.775,6.475,149.115
C03094=1140.068,56.226,-52.021,-179.772,6.476,149.114
C03095=1140.064,56.476,-52.037,-179.770,6.477,149.114
C03096=1140.059,56.724,-52.053,-179.766,6.478,149.113
C03097=1140.054,56.975,-52.069,-179.764,6.479,149.113
C03098=1140.048,57.224,-52.085,-179.762,6.481,149.112
C03099=1140.043,57.473,-52.101,-179.758,6.482,149.112
C03100=1140.039,57.723,-52.117,-179.756,6.483,149.111
C03101=1140.033,57.972,-52.133,-179.753,6.485,149.111
C03102=1140.029,58.222,-52.149,-179.751,6.485,149.110
C03103=1140.023,58.471,-52.165,-179.748,6.487,149.110
C03104=1140.018,58.720,-52.181,-179.745,6.488,149.109
C03105=1140.013,58.970,-52.197,-179.743,6.489,149.109
C03106=1140.009,59.219,-52.212,-179.740,6.490,149.108
C03107=1140.004,59.469,-52.229,-179.738,6.491,149.108
C03108=1139.999,59.718,-52.244,-179.735,6.493,149.107
C03109=1139.994,59.967,-52.261,-179.732,6.494,149.106
C03110=1139.989,60.217,-52.277,-179.730,6.495,149.106
C03111=1139.984,60.466,-52.293,-179.727,6.497,149.106
C03112=1139.979,60.716,-52.309,-179.724,6.497,149.105
C03113=1139.974,60.965,-52.325,-179.721,6.499,149.105
C03114=1139.969,61.215,-52.342,-179.719,6.500,149.104
C03115=1139.963,61.464,-52.357,-179.716,6.501,149.104
C03116=1139.959,61.714,-52.374,-179.713,6.503,149.103
C03117=1139.953,61.963,-52.390,-179.711,6.503,149.103
C03118=1139.949,62.213,-52.406,-179.708,6.505,149.102
C03119=1139.944,62.462,-52.423,-179.705,6.506,149.101
C03120=1139.939,62.712,-52.439,-179.703,6.507,149.101
C03121=1139.934,62.960,-52.455,-179.700,6.509,149.101
C03122=1139.929,63.211,-52.471,-179.697,6.510,149.100
C03123=1139.924,63.459,-52.487,-179.695,6.511,149.099
C03124=1139.919,63.709,-52.503,-179.692,6.513,149.099
C03125=1139.914,63.958,-52.519,-179.689,6.514,149.099
C03126=1139.910,64.208,-52.536,-179.687,6.515,149.098
C03127=1139.904,64.457,-52.552,-179.684,6.516,149.097
C03128=1139.899,64.707,-52.569,-179.682,6.517,149.097
C03129=1139.894,64.956,-52.585,-179.679,6.519,149.096
C03130=1139.889,65.206,-52.601,-179.676,6.520,149.096
C03131=1139.884,65.455,-52.618,-179.674,6.521,149.096
C03132=1139.879,65.705,-52.633,-179.671,6.523,149.095
C03133=1139.874,65.953,-52.650,-179.668,6.524,149.094
C03134=1139.870,66.203,-52.666,-179.666,6.525,149.094
C03135=1139.864,66.453,-52.683,-179.663,6.526,149.094
C03136=1139.859,66.702,-52.699,-179.660,6.528,149.093
C03137=1139.855,66.952,-52.716,-179.657,6.529,149.092
C03138=1139.850,67.200,-52.732,-179.655,6.530,149.092
C03139=1139.845,67.451,-52.748,-179.652,6.532,149.092
C03140=1139.839,67.700,-52.765,-179.649,6.532,149.091
C03141=1139.835,67.949,-52.782,-179.646,6.534,149.090
C03142=1139.829,68.198,-52.798,-179.644,6.536,149.090
C03143=1139.825,68.448,-52.814,-179.642,6.537,149.090
C03144=1139.820,68.697,-52.831,-179.638,6.538,149.089
C03145=1139.814,68.947,-52.848,-179.636,6.539,149.089
C03146=1139.810,69.196,-52.864,-179.633,6.540,149.088
C03147=1139.805,69.445,-52.881,-179.630,6.542,149.087
C03148=1139.800,69.695,-52.897,-179.627,6.543,149.087
C03149=1139.795,69.945,-52.914,-179.625,6.544,149.087
C03150=1139.790,70.193,-52.930,-179.623,6.546,149.086
C03151=1139.785,70.443,-52.947,-179.619,6.547,149.085
C03152=1139.780,70.693,-52.964,-179.617,6.548,149.085
C03153=1139.775,70.942,-52.980,-179.614,6.550,149.085
C03154=1139.770,71.191,-52.997,-179.612,6.551,149.084
C03155=1139.765,71.440,-53.013,-179.608,6.552,149.084
C03156=1139.760,71.690,-53.030,-179.606,6.553,149.083
C03157=1139.755,71.940,-53.047,-179.604,6.555,149.083
C03158=1139.750,72.188,-53.063,-179.600,6.556,149.082
C03159=1139.745,72.438,-53.080,-179.598,6.557,149.082
C03160=1139.741,72.688,-53.097,-179.595,6.559,149.081
C03161=1139.735,72.937,-53.114,-179.593,6.560,149.081
C03162=1139.730,73.186,-53.130,-179.590,6.561,149.080
C03163=1139.726,73.436,-53.147,-179.587,6.563,149.080
C03164=1139.720,73.685,-53.164,-179.585,6.564,149.079
C03165=1139.715,73.934,-53.181,-179.582,6.566,149.079
C03166=1139.711,74.184,-53.197,-179.579,6.566,149.078
C03167=1139.706,74.434,-53.215,-179.576,6.568,149.078
C03168=1139.701,74.682,-53.231,-179.574,6.570,149.077
C03169=1139.695,74.932,-53.248,-179.572,6.571,149.077
C03170=1139.691,75.182,-53.265,-179.568,6.572,149.076
C03171=1139.686,75.431,-53.281,-179.566,6.573,149.076
C03172=1139.681,75.680,-53.298,-179.563,6.575,149.075
C03173=1139.676,75.930,-53.315,-179.561,6.576,149.075
C03174=1139.671,76.179,-53.333,-179.557,6.577,149.074
C03175=1139.666,76.428,-53.349,-179.555,6.579,149.074
C03176=1139.661,76.678,-53.367,-179.552,6.581,149.073
C03177=1139.657,76.927,-53.383,-179.550,6.581,149.073
C03178=1139.651,77.177,-53.400,-179.547,6.583,149.072
C03179=1139.646,77.426,-53.417,-179.544,6.584,149.072
C03180=1139.641,77.675,-53.434,-179.542,6.585,149.071
C03181=1139.637,77.925,-53.451,-179.539,6.587,149.071
C03182=1139.632,78.174,-53.469,-179.536,6.588,149.070
C03183=1139.627,78.423,-53.485,-179.533,6.590,149.070
C03184=1139.621,78.673,-53.502,-179.531,6.591,149.069
C03185=1139.617,78.922,-53.519,-179.528,6.592,149.069
C03186=1139.611,79.191,-53.538,-179.525,6.594,149.068
C03187=1139.606,79.459,-53.555,-179.522,6.595,149.068
C03188=1139.601,79.728,-53.574,-179.519,6.597,149.068
C03189=1139.595,79.995,-53.593,-179.516,6.598,149.067
C03190=1139.591,80.245,-53.610,-179.513,6.600,149.066
C03191=1139.585,80.495,-53.627,-179.511,6.602,149.066
C03192=1139.581,80.744,-53.644,-179.508,6.602,149.065
C03193=1139.576,80.993,-53.662,-179.505,6.604,149.065
C03194=1139.570,81.242,-53.679,-179.503,6.605,149.065
C03195=1139.566,81.492,-53.695,-179.500,6.607,149.064
C03196=1139.561,81.741,-53.713,-179.498,6.608,149.064
C03197=1139.556,81.990,-53.730,-179.494,6.609,149.063
C03198=1139.551,82.240,-53.747,-179.492,6.611,149.063
C03199=1139.546,82.489,-53.765,-179.489,6.613,149.062
C03200=1139.542,82.739,-53.782,-179.487,6.613,149.062
C03201=1139.536,82.988,-53.799,-179.484,6.615,149.061
C03202=1139.531,83.237,-53.817,-179.481,6.616,149.061
C03203=1139.527,83.487,-53.833,-179.478,6.618,149.060
C03204=1139.522,83.736,-53.851,-179.475,6.620,149.060
C03205=1139.517,83.985,-53.868,-179.473,6.621,149.059
C03206=1139.512,84.235,-53.885,-179.470,6.622,149.059
C03207=1139.507,84.484,-53.903,-179.467,6.624,149.058
C03208=1139.502,84.734,-53.921,-179.464,6.625,149.058
C03209=1139.497,84.982,-53.938,-179.462,6.627,149.057
C03210=1139.492,85.232,-53.955,-179.459,6.627,149.057
C03211=1139.487,85.481,-53.973,-179.456,6.629,149.056
C03212=1139.482,85.731,-53.989,-179.454,6.631,149.056
C03213=1139.478,85.980,-54.007,-179.451,6.632,149.056
C03214=1139.472,86.230,-54.025,-179.448,6.634,149.055
C03215=1139.467,86.479,-54.043,-179.446,6.634,149.054
C03216=1139.463,86.728,-54.059,-179.443,6.636,149.054
C03217=1139.458,86.978,-54.077,-179.440,6.638,149.054
C03218=1139.453,87.227,-54.095,-179.437,6.639,149.053
C03219=1139.448,87.477,-54.113,-179.435,6.641,149.053
C03220=1139.443,87.726,-54.129,-179.432,6.642,149.052
C03221=1139.438,87.975,-54.147,-179.429,6.643,149.052
C03222=1139.434,88.224,-54.165,-179.426,6.645,149.051
C03223=1139.428,88.474,-54.182,-179.424,6.647,149.051
C03224=1139.423,88.723,-54.200,-179.421,6.648,149.050
C03225=1139.418,88.972,-54.217,-179.418,6.650,149.050
C03226=1139.413,89.221,-54.235,-179.416,6.650,149.049
C03227=1139.409,89.470,-54.253,-179.413,6.652,149.049
C03228=1139.403,89.720,-54.270,-179.410,6.654,149.048
C03229=1139.398,89.969,-54.288,-179.407,6.655,149.048
C03230=1139.393,90.219,-54.306,-179.404,6.657,149.047
C03231=1139.389,90.468,-54.323,-179.401,6.658,149.047
C03232=1139.384,90.717,-54.341,-179.399,6.659,149.047
C03233=1139.379,90.966,-54.359,-179.397,6.661,149.046
C03234=1139.374,91.216,-54.377,-179.394,6.663,149.046
C03235=1139.369,91.465,-54.394,-179.391,6.664,149.045
C03236=1139.364,91.715,-54.412,-179.388,6.666,149.045
C03237=1139.360,91.964,-54.430,-179.385,6.667,149.044
C03238=1139.355,92.214,-54.448,-179.383,6.668,149.044
C03239=1139.350,92.463,-54.465,-179.380,6.670,149.043
C03240=1139.346,92.712,-54.483,-179.377,6.671,149.043
C03241=1139.341,92.961,-54.501,-179.374,6.673,149.042
C03242=1139.336,93.211,-54.519,-179.372,6.674,149.042
C03243=1139.331,93.460,-54.537,-179.369,6.676,149.042
C03244=1139.326,93.710,-54.554,-179.366,6.678,149.041
C03245=1139.321,93.959,-54.572,-179.364,6.679,149.041
C03246=1139.316,94.208,-54.590,-179.361,6.680,149.040
C03247=1139.311,94.457,-54.608,-179.358,6.682,149.040
C03248=1139.306,94.706,-54.626,-179.355,6.683,149.039
C03249=1139.301,94.955,-54.644,-179.352,6.685,149.039
C03250=1139.296,95.205,-54.662,-179.350,6.687,149.038
C03251=1139.291,95.454,-54.679,-179.347,6.688,149.038
C03252=1139.287,95.704,-54.697,-179.344,6.690,149.038
C03253=1139.282,95.954,-54.715,-179.342,6.690,149.037
C03254=1139.277,96.203,-54.733,-179.339,6.692,149.036
C03255=1139.272,96.452,-54.751,-179.336,6.694,149.036
C03256=1139.267,96.701,-54.769,-179.333,6.695,149.036
C03257=1139.262,96.950,-54.787,-179.331,6.697,149.035
C03258=1139.257,97.199,-54.805,-179.328,6.699,149.035
C03259=1139.252,97.449,-54.823,-179.325,6.700,149.034
C03260=1139.247,97.699,-54.842,-179.322,6.702,149.034
C03261=1139.242,97.948,-54.860,-179.320,6.703,149.033
C03262=1139.237,98.197,-54.878,-179.317,6.704,149.033
C03263=1139.232,98.446,-54.896,-179.314,6.706,149.032
C03264=1139.227,98.695,-54.914,-179.312,6.708,149.032
C03265=1139.223,98.945,-54.932,-179.309,6.709,149.032
C03266=1139.218,99.195,-54.950,-179.306,6.711,149.031
C03267=1139.213,99.444,-54.968,-179.303,6.712,149.031
C03268=1139.208,99.693,-54.986,-179.300,6.714,149.030
C03269=1139.203,99.942,-55.006,-179.297,6.716,149.030
C03270=1139.198,100.191,-55.024,-179.295,6.717,149.029
C03271=1139.193,100.440,-55.042,-179.292,6.719,149.029
C03272=1139.189,100.690,-55.060,-179.290,6.720,149.028
C03273=1139.184,100.939,-55.078,-179.287,6.721,149.028
C03274=1139.179,101.188,-55.096,-179.284,6.723,149.027
C03275=1139.174,101.437,-55.114,-179.281,6.725,149.027
C03276=1139.169,101.686,-55.133,-179.278,6.726,149.027
C03277=1139.165,101.936,-55.152,-179.276,6.728,149.026
C03278=1139.160,102.185,-55.170,-179.273,6.730,149.026
C03279=1139.155,102.435,-55.188,-179.270,6.731,149.025
C03280=1139.149,102.684,-55.206,-179.268,6.733,149.025
C03281=1139.145,102.933,-55.225,-179.264,6.734,149.024
C03282=1139.140,103.183,-55.243,-179.262,6.736,149.024
C03283=1139.135,103.432,-55.261,-179.259,6.738,149.023
C03284=1139.130,103.681,-55.279,-179.256,6.739,149.023
C03285=1139.126,103.930,-55.299,-179.254,6.740,149.023
C03286=1139.121,104.180,-55.317,-179.251,6.742,149.022
C03287=1139.116,104.429,-55.335,-179.249,6.744,149.022
C03288=1139.110,104.678,-55.353,-179.246,6.745,149.021
C03289=1139.106,104.928,-55.372,-179.243,6.747,149.021
C03290=1139.101,105.196,-55.392,-179.240,6.748,149.020
C03291=1139.095,105.464,-55.412,-179.236,6.751,149.020
C03292=1139.090,105.733,-55.431,-179.234,6.752,149.020
C03293=1139.085,106.001,-55.452,-179.231,6.754,149.019
C03294=1139.080,106.250,-55.470,-179.228,6.755,149.019
C03295=1139.075,106.500,-55.488,-179.225,6.757,149.018
C03296=1139.070,106.748,-55.508,-179.222,6.759,149.018
C03297=1139.066,106.998,-55.526,-179.220,6.760,149.017
C03298=1139.061,107.247,-55.545,-179.217,6.762,149.017
C03299=1139.055,107.496,-55.563,-179.214,6.764,149.016
C03300=1139.051,107.746,-55.582,-179.211,6.765,149.016
C03301=1139.047,107.995,-55.600,-179.208,6.767,149.015
C03302=1139.042,108.245,-55.619,-179.205,6.768,149.015
C03303=1139.037,108.494,-55.638,-179.203,6.770,149.015
C03304=1139.031,108.743,-55.656,-179.200,6.772,149.014
C03305=1139.027,108.992,-55.675,-179.197,6.773,149.014
C03306=1139.022,109.241,-55.693,-179.195,6.775,149.013
C03307=1139.017,109.490,-55.713,-179.192,6.777,149.013
C03308=1139.013,109.740,-55.731,-179.189,6.779,149.013
C03309=1139.007,109.989,-55.750,-179.186,6.780,149.012
C03310=1139.002,110.238,-55.768,-179.184,6.781,149.012
C03311=1138.998,110.488,-55.788,-179.181,6.783,149.011
C03312=1138.993,110.736,-55.807,-179.178,6.784,149.011
C03313=1138.988,110.987,-55.826,-179.176,6.786,149.010
C03314=1138.983,111.235,-55.844,-179.173,6.787,149.010
C03315=1138.978,111.485,-55.863,-179.170,6.789,149.009
C03316=1138.974,111.734,-55.882,-179.167,6.791,149.009
C03317=1138.968,111.983,-55.901,-179.165,6.792,149.009
C03318=1138.964,112.233,-55.920,-179.162,6.794,149.008
C03319=1138.959,112.481,-55.939,-179.159,6.796,149.008
C03320=1138.955,112.731,-55.958,-179.156,6.798,149.007
C03321=1138.949,112.980,-55.977,-179.154,6.799,149.007
C03322=1138.945,113.229,-55.995,-179.151,6.801,149.007
C03323=1138.940,113.478,-56.015,-179.148,6.803,149.006
C03324=1138.935,113.728,-56.033,-179.145,6.805,149.006
C03325=1138.930,113.977,-56.053,-179.142,6.806,149.005
C03326=1138.926,114.226,-56.071,-179.139,6.808,149.005
C03327=1138.920,114.476,-56.090,-179.136,6.810,149.004
C03328=1138.915,114.725,-56.109,-179.134,6.811,149.004
C03329=1138.911,114.974,-56.129,-179.131,6.813,149.004
C03330=1138.906,115.223,-56.148,-179.128,6.815,149.003
C03331=1138.901,115.473,-56.166,-179.125,6.816,149.003
C03332=1138.896,115.722,-56.185,-179.123,6.818,149.002
C03333=1138.891,115.971,-56.205,-179.120,6.820,149.002
C03334=1138.887,116.220,-56.224,-179.117,6.822,149.002
C03335=1138.882,116.469,-56.243,-179.114,6.823,149.001
C03336=1138.876,116.719,-56.262,-179.112,6.825,149.001
C03337=1138.872,116.968,-56.281,-179.109,6.827,149.000
C03338=1138.867,117.217,-56.300,-179.106,6.828,149.000
C03339=1138.862,117.466,-56.320,-179.104,6.830,148.999
C03340=1138.858,117.715,-56.339,-179.101,6.832,148.999
C03341=1138.853,117.965,-56.358,-179.098,6.833,148.999
C03342=1138.848,118.213,-56.378,-179.095,6.835,148.998
C03343=1138.844,118.463,-56.397,-179.092,6.836,148.998
C03344=1138.838,118.712,-56.416,-179.089,6.838,148.997
C03345=1138.833,118.962,-56.435,-179.087,6.840,148.997
C03346=1138.829,119.211,-56.454,-179.084,6.841,148.996
C03347=1138.824,119.460,-56.473,-179.081,6.843,148.996
C03348=1138.819,119.709,-56.493,-179.078,6.845,148.996
C03349=1138.814,119.958,-56.512,-179.075,6.847,148.995
C03350=1138.810,120.208,-56.531,-179.072,6.849,148.995
C03351=1138.804,120.456,-56.551,-179.070,6.851,148.994
C03352=1138.800,120.706,-56.570,-179.067,6.852,148.994
C03353=1138.795,120.956,-56.590,-179.064,6.854,148.994
C03354=1138.790,121.204,-56.609,-179.062,6.856,148.993
C03355=1138.786,121.454,-56.628,-179.059,6.857,148.993
C03356=1138.780,121.703,-56.648,-179.056,6.859,148.992
C03357=1138.776,121.952,-56.668,-179.053,6.861,148.992
C03358=1138.771,122.201,-56.688,-179.051,6.862,148.992
C03359=1138.766,122.450,-56.706,-179.048,6.864,148.991
C03360=1138.762,122.699,-56.726,-179.045,6.866,148.991
C03361=1138.757,122.949,-56.746,-179.042,6.868,148.990
C03362=1138.752,123.198,-56.765,-179.039,6.870,148.990
C03363=1138.747,123.447,-56.785,-179.036,6.872,148.990
C03364=1138.742,123.697,-56.804,-179.034,6.873,148.989
C03365=1138.737,123.945,-56.824,-179.031,6.875,148.989
C03366=1138.733,124.194,-56.843,-179.028,6.877,148.988
C03367=1138.728,124.444,-56.863,-179.026,6.878,148.988
C03368=1138.723,124.693,-56.882,-179.023,6.880,148.988
C03369=1138.718,124.942,-56.902,-179.020,6.882,148.987
C03370=1138.714,125.192,-56.922,-179.017,6.884,148.987
C03371=1138.708,125.440,-56.942,-179.015,6.885,148.986
C03372=1138.704,125.690,-56.961,-179.011,6.888,148.986
C03373=1138.699,125.939,-56.981,-179.009,6.889,148.986
C03374=1138.694,126.188,-57.000,-179.006,6.891,148.985
C03375=1138.689,126.437,-57.021,-179.003,6.893,148.985
C03376=1138.685,126.686,-57.040,-179.000,6.895,148.984
C03377=1138.680,126.936,-57.059,-178.998,6.896,148.984
C03378=1138.675,127.184,-57.079,-178.995,6.898,148.984
C03379=1138.671,127.434,-57.099,-178.992,6.900,148.983
C03380=1138.666,127.683,-57.119,-178.990,6.901,148.983
C03381=1138.661,127.932,-57.139,-178.986,6.904,148.982
C03382=1138.656,128.181,-57.158,-178.983,6.905,148.982
C03383=1138.651,128.431,-57.178,-178.981,6.907,148.982
C03384=1138.647,128.680,-57.198,-178.978,6.909,148.981
C03385=1138.642,128.928,-57.218,-178.975,6.911,148.981
C03386=1138.637,129.177,-57.238,-178.973,6.912,148.980
C03387=1138.632,129.427,-57.258,-178.970,6.914,148.980
C03388=1138.628,129.677,-57.277,-178.967,6.916,148.980
C03389=1138.622,129.925,-57.298,-178.964,6.918,148.979
C03390=1138.617,130.175,-57.317,-178.961,6.920,148.979
C03391=1138.613,130.424,-57.338,-178.958,6.922,148.978
C03392=1138.608,130.673,-57.358,-178.956,6.923,148.978
C03393=1138.604,130.922,-57.378,-178.953,6.925,148.978
C03394=1138.599,131.191,-57.399,-178.950,6.927,148.977
C03395=1138.593,131.460,-57.421,-178.947,6.929,148.977
C03396=1138.588,131.728,-57.442,-178.944,6.931,148.977
C03397=1138.583,131.997,-57.464,-178.941,6.933,148.976
C03398=1138.577,132.246,-57.483,-178.938,6.935,148.976
C03399=1138.573,132.495,-57.504,-178.935,6.937,148.975
C03400=1138.569,132.744,-57.524,-178.933,6.938,148.975
C03401=1138.564,132.993,-57.544,-178.930,6.940,148.975
C03402=1138.559,133.242,-57.564,-178.927,6.943,148.974
C03403=1138.555,133.492,-57.584,-178.924,6.944,148.974
C03404=1138.549,133.740,-57.604,-178.921,6.946,148.973
C03405=1138.544,133.989,-57.625,-178.918,6.948,148.973
C03406=1138.540,134.239,-57.644,-178.916,6.949,148.973
C03407=1138.535,134.488,-57.665,-178.912,6.952,148.972
C03408=1138.530,134.737,-57.685,-178.910,6.954,148.972
C03409=1138.525,134.986,-57.705,-178.907,6.956,148.972
C03410=1138.521,135.235,-57.726,-178.905,6.957,148.971
C03411=1138.516,135.484,-57.745,-178.902,6.959,148.971
C03412=1138.511,135.733,-57.766,-178.899,6.961,148.970
C03413=1138.507,135.982,-57.786,-178.896,6.963,148.970
C03414=1138.501,136.231,-57.807,-178.893,6.965,148.970
C03415=1138.497,136.481,-57.827,-178.891,6.967,148.969
C03416=1138.492,136.730,-57.847,-178.888,6.968,148.969
C03417=1138.487,136.979,-57.868,-178.885,6.970,148.969
C03418=1138.483,137.228,-57.888,-178.882,6.973,148.968
C03419=1138.478,137.478,-57.908,-178.879,6.974,148.968
C03420=1138.473,137.727,-57.928,-178.876,6.976,148.967
C03421=1138.468,137.976,-57.949,-178.874,6.978,148.967
C03422=1138.464,138.225,-57.970,-178.871,6.980,148.967
C03423=1138.459,138.474,-57.990,-178.868,6.982,148.966
C03424=1138.454,138.724,-58.010,-178.865,6.984,148.966
C03425=1138.449,138.972,-58.030,-178.863,6.986,148.966
C03426=1138.444,139.221,-58.051,-178.860,6.987,148.965
C03427=1138.439,139.470,-58.072,-178.857,6.989,148.965
C03428=1138.435,139.719,-58.092,-178.854,6.992,148.964
C03429=1138.430,139.968,-58.112,-178.851,6.993,148.964
C03430=1138.425,140.217,-58.133,-178.849,6.995,148.964
C03431=1138.421,140.466,-58.154,-178.846,6.997,148.963
C03432=1138.416,140.715,-58.174,-178.843,7.000,148.963
C03433=1138.411,140.964,-58.195,-178.840,7.001,148.963
C03434=1138.407,141.213,-58.215,-178.838,7.003,148.962
C03435=1138.402,141.463,-58.236,-178.835,7.005,148.962
C03436=1138.397,141.712,-58.256,-178.831,7.007,148.962
C03437=1138.392,141.962,-58.277,-178.829,7.009,148.961
C03438=1138.387,142.210,-58.297,-178.826,7.011,148.961
C03439=1138.384,142.459,-58.319,-178.823,7.012,148.960
C03440=1138.379,142.709,-58.340,-178.820,7.015,148.960
C03441=1138.374,142.958,-58.360,-178.818,7.017,148.960
C03442=1138.369,143.207,-58.381,-178.815,7.019,148.959
C03443=1138.364,143.456,-58.401,-178.812,7.020,148.959
C03444=1138.359,143.705,-58.422,-178.810,7.022,148.959
C03445=1138.355,143.954,-58.443,-178.806,7.024,148.958
C03446=1138.350,144.203,-58.464,-178.804,7.026,148.958
C03447=1138.345,144.452,-58.484,-178.801,7.028,148.958
C03448=1138.340,144.702,-58.505,-178.798,7.030,148.957
C03449=1138.336,144.951,-58.525,-178.795,7.032,148.957
C03450=1138.330,145.200,-58.546,-178.793,7.034,148.957
C03451=1138.326,145.448,-58.568,-178.790,7.036,148.956
C03452=1138.321,145.697,-58.588,-178.787,7.038,148.956
C03453=1138.317,145.947,-58.609,-178.784,7.040,148.955
C03454=1138.312,146.196,-58.630,-178.781,7.042,148.955
C03455=1138.307,146.446,-58.651,-178.778,7.043,148.955
C03456=1138.303,146.694,-58.672,-178.776,7.046,148.955
C03457=1138.298,146.943,-58.693,-178.773,7.048,148.954
C03458=1138.293,147.192,-58.714,-178.770,7.050,148.954
C03459=1138.288,147.441,-58.735,-178.767,7.051,148.953
C03460=1138.284,147.690,-58.756,-178.764,7.054,148.953
C03461=1138.279,147.940,-58.777,-178.761,7.056,148.953
C03462=1138.274,148.189,-58.798,-178.759,7.057,148.952
C03463=1138.270,148.438,-58.818,-178.756,7.060,148.952
C03464=1138.265,148.686,-58.840,-178.753,7.062,148.952
C03465=1138.260,148.936,-58.861,-178.750,7.064,148.951
C03466=1138.255,149.185,-58.881,-178.747,7.066,148.951
C03467=1138.251,149.434,-58.903,-178.744,7.068,148.951
C03468=1138.246,149.683,-58.924,-178.742,7.070,148.950
C03469=1138.241,149.932,-58.945,-178.740,7.072,148.950
C03470=1138.237,150.181,-58.966,-178.736,7.074,148.950
C03471=1138.231,150.430,-58.987,-178.733,7.076,148.949
C03472=1138.227,150.678,-59.008,-178.731,7.078,148.949
C03473=1138.223,150.928,-59.030,-178.727,7.080,148.949
C03474=1138.217,151.178,-59.051,-178.725,7.082,148.948
C03475=1138.213,151.426,-59.072,-178.723,7.084,148.948
C03476=1138.208,151.675,-59.093,-178.719,7.086,148.948
C03477=1138.203,151.924,-59.114,-178.717,7.088,148.947
C03478=1138.199,152.174,-59.136,-178.714,7.090,148.947
C03479=1138.194,152.423,-59.158,-178.710,7.092,148.946
C03480=1138.189,152.671,-59.178,-178.708,7.094,148.946
C03481=1138.185,152.920,-59.200,-178.706,7.096,148.946
C03482=1138.180,153.170,-59.221,-178.702,7.099,148.946
C03483=1138.175,153.419,-59.243,-178.700,7.100,148.945
C03484=1138.170,153.668,-59.264,-178.697,7.102,148.945
C03485=1138.166,153.916,-59.285,-178.695,7.104,148.945
C03486=1138.161,154.166,-59.306,-178.691,7.107,148.944
C03487=1138.156,154.415,-59.328,-178.689,7.108,148.944
C03488=1138.151,154.664,-59.349,-178.685,7.111,148.944
C03489=1138.147,154.914,-59.371,-178.683,7.113,148.943
C03490=1138.142,155.162,-59.392,-178.680,7.115,148.943
C03491=1138.137,155.411,-59.413,-178.677,7.117,148.943
C03492=1138.133,155.660,-59.434,-178.674,7.119,148.942
C03493=1138.128,155.909,-59.456,-178.672,7.121,148.942
C03494=1138.123,156.158,-59.477,-178.669,7.123,148.942
C03495=1138.118,156.407,-59.499,-178.666,7.125,148.941
C03496=1138.114,156.656,-59.521,-178.663,7.127,148.941
C03497=1138.109,156.905,-59.543,-178.660,7.129,148.941
C03498=1138.105,157.174,-59.566,-178.657,7.131,148.940
C03499=1138.099,157.443,-59.589,-178.654,7.134,148.940
C03500=1138.094,157.712,-59.612,-178.651,7.136,148.940
C03501=1138.089,157.981,-59.636,-178.648,7.138,148.939
C03502=1138.084,158.230,-59.657,-178.645,7.141,148.939
C03503=1138.080,158.480,-59.679,-178.642,7.142,148.939
C03504=1138.075,158.728,-59.700,-178.640,7.144,148.938
C03505=1138.070,158.977,-59.722,-178.637,7.147,148.938
C03506=1138.066,159.226,-59.744,-178.634,7.149,148.938
C03507=1138.061,159.475,-59.766,-178.632,7.150,148.937
C03508=1138.056,159.724,-59.787,-178.628,7.153,148.937
C03509=1138.051,159.974,-59.809,-178.626,7.155,148.937
C03510=1138.046,160.222,-59.831,-178.623,7.158,148.936
C03511=1138.042,160.472,-59.853,-178.620,7.159,148.936
C03512=1138.037,160.720,-59.874,-178.617,7.161,148.936
C03513=1138.033,160.970,-59.896,-178.614,7.164,148.936
C03514=1138.028,161.218,-59.918,-178.612,7.166,148.935
C03515=1138.023,161.467,-59.940,-178.609,7.167,148.935
C03516=1138.019,161.716,-59.962,-178.606,7.170,148.934
C03517=1138.014,161.965,-59.983,-178.603,7.172,148.934
C03518=1138.010,162.214,-60.006,-178.600,7.174,148.934
C03519=1138.005,162.463,-60.026,-178.597,7.176,148.934
C03520=1138.001,162.713,-60.049,-178.595,7.178,148.933
C03521=1137.995,162.962,-60.071,-178.592,7.181,148.933
C03522=1137.991,163.211,-60.093,-178.589,7.182,148.933
C03523=1137.986,163.459,-60.115,-178.586,7.185,148.932
C03524=1137.981,163.708,-60.137,-178.584,7.187,148.932
C03525=1137.977,163.957,-60.159,-178.580,7.190,148.932
C03526=1137.972,164.206,-60.181,-178.578,7.191,148.931
C03527=1137.968,164.455,-60.203,-178.575,7.193,148.931
C03528=1137.963,164.704,-60.224,-178.572,7.196,148.931
C03529=1137.958,164.953,-60.247,-178.569,7.198,148.931
C03530=1137.953,165.202,-60.269,-178.566,7.200,148.930
C03531=1137.949,165.451,-60.291,-178.564,7.202,148.930
C03532=1137.944,165.700,-60.312,-178.561,7.204,148.930
C03533=1137.940,165.949,-60.335,-178.558,7.206,148.929
C03534=1137.935,166.198,-60.358,-178.555,7.208,148.929
C03535=1137.930,166.447,-60.380,-178.552,7.211,148.929
C03536=1137.926,166.696,-60.402,-178.550,7.213,148.928
C03537=1137.921,166.945,-60.423,-178.546,7.215,148.928
C03538=1137.916,167.195,-60.446,-178.544,7.217,148.928
C03539=1137.911,167.443,-60.468,-178.541,7.220,148.928
C03540=1137.907,167.692,-60.490,-178.538,7.222,148.927
C03541=1137.902,167.941,-60.512,-178.536,7.224,148.927
C03542=1137.897,168.190,-60.535,-178.533,7.226,148.927
C03543=1137.892,168.439,-60.556,-178.530,7.228,148.926
C03544=1137.888,168.688,-60.579,-178.527,7.231,148.926
C03545=1137.884,168.937,-60.601,-178.524,7.232,148.926
C03546=1137.879,169.186,-60.623,-178.521,7.235,148.925
C03547=1137.875,169.435,-60.646,-178.519,7.237,148.925
C03548=1137.870,169.683,-60.668,-178.516,7.240,148.925
C03549=1137.865,169.933,-60.691,-178.513,7.241,148.925
C03550=1137.861,170.182,-60.713,-178.510,7.244,148.924
C03551=1137.855,170.431,-60.736,-178.507,7.246,148.924
C03552=1137.851,170.680,-60.758,-178.505,7.248,148.924
C03553=1137.846,170.928,-60.780,-178.502,7.251,148.924
C03554=1137.841,171.178,-60.803,-178.499,7.252,148.923
C03555=1137.837,171.426,-60.825,-178.496,7.255,148.923
C03556=1137.832,171.675,-60.847,-178.494,7.257,148.923
C03557=1137.827,171.925,-60.870,-178.490,7.259,148.922
C03558=1137.823,172.173,-60.893,-178.488,7.261,148.922
C03559=1137.818,172.422,-60.915,-178.485,7.264,148.922
C03560=1137.814,172.671,-60.938,-178.482,7.266,148.921
C03561=1137.810,172.920,-60.960,-178.479,7.268,148.921
C03562=1137.804,173.169,-60.983,-178.477,7.270,148.921
C03563=1137.800,173.418,-61.005,-178.473,7.273,148.921
C03564=1137.795,173.667,-61.028,-178.471,7.275,148.920
C03565=1137.791,173.916,-61.050,-178.468,7.277,148.920
C03566=1137.786,174.165,-61.073,-178.465,7.279,148.920
C03567=1137.782,174.414,-61.095,-178.462,7.282,148.920
C03568=1137.776,174.662,-61.118,-178.459,7.284,148.919
C03569=1137.772,174.911,-61.141,-178.456,7.286,148.919
C03570=1137.767,175.161,-61.164,-178.454,7.288,148.919
C03571=1137.763,175.409,-61.186,-178.451,7.291,148.918
C03572=1137.758,175.658,-61.209,-178.448,7.293,148.918
C03573=1137.754,175.907,-61.231,-178.445,7.296,148.918
C03574=1137.749,176.156,-61.255,-178.442,7.297,148.918
C03575=1137.744,176.405,-61.276,-178.440,7.300,148.917
C03576=1137.739,176.654,-61.300,-178.437,7.302,148.917
C03577=1137.735,176.903,-61.323,-178.434,7.304,148.917
C03578=1137.730,177.152,-61.345,-178.431,7.306,148.917
C03579=1137.725,177.401,-61.368,-178.428,7.309,148.916
C03580=1137.721,177.649,-61.391,-178.426,7.311,148.916
C03581=1137.717,177.898,-61.414,-178.423,7.314,148.916
C03582=1137.712,178.148,-61.436,-178.420,7.315,148.915
C03583=1137.708,178.397,-61.460,-178.417,7.318,148.915
C03584=1137.702,178.645,-61.483,-178.414,7.320,148.915
C03585=1137.698,178.894,-61.505,-178.412,7.323,148.915
C03586=1137.694,179.143,-61.529,-178.408,7.325,148.914
C03587=1137.689,179.392,-61.551,-178.406,7.327,148.914
C03588=1137.685,179.641,-61.574,-178.403,7.330,148.914
C03589=1137.679,179.890,-61.597,-178.400,7.332,148.913
C03590=1137.675,180.139,-61.621,-178.397,7.335,148.913
C03591=1137.671,180.387,-61.643,-178.394,7.336,148.913
C03592=1137.666,180.636,-61.667,-178.392,7.339,148.913
C03593=1137.661,180.886,-61.689,-178.389,7.341,148.913
C03594=1137.657,181.135,-61.712,-178.386,7.343,148.912
C03595=1137.652,181.383,-61.735,-178.383,7.346,148.912
C03596=1137.647,181.632,-61.758,-178.380,7.348,148.912
C03597=1137.643,181.881,-61.781,-178.377,7.351,148.912
C03598=1137.638,182.130,-61.805,-178.375,7.353,148.911
C03599=1137.634,182.379,-61.828,-178.372,7.356,148.911
C03600=1137.629,182.628,-61.851,-178.369,7.357,148.911
C03601=1137.625,182.877,-61.874,-178.366,7.360,148.911
C03602=1137.620,183.146,-61.899,-178.363,7.363,148.910
C03603=1137.614,183.416,-61.924,-178.360,7.365,148.910
C03604=1137.609,183.685,-61.950,-178.357,7.367,148.910
C03605=1137.604,183.955,-61.975,-178.354,7.370,148.909
C03606=1137.600,184.204,-61.998,-178.351,7.372,148.909
C03607=1137.595,184.453,-62.021,-178.349,7.375,148.909
C03608=1137.591,184.702,-62.044,-178.345,7.377,148.909
C03609=1137.586,184.951,-62.068,-178.343,7.380,148.908
C03610=1137.581,185.200,-62.091,-178.340,7.382,148.908
C03611=1137.577,185.449,-62.114,-178.337,7.385,148.908
C03612=1137.573,185.697,-62.138,-178.334,7.386,148.908
C03613=1137.568,185.946,-62.161,-178.332,7.389,148.907
C03614=1137.563,186.195,-62.185,-178.328,7.392,148.907
C03615=1137.559,186.444,-62.208,-178.326,7.394,148.907
C03616=1137.553,186.692,-62.231,-178.323,7.396,148.907
C03617=1137.549,186.941,-62.254,-178.320,7.398,148.907
C03618=1137.544,187.190,-62.278,-178.317,7.401,148.906
C03619=1137.540,187.439,-62.302,-178.314,7.404,148.906
C03620=1137.535,187.688,-62.325,-178.312,7.406,148.906
C03621=1137.530,187.937,-62.348,-178.308,7.408,148.905
C03622=1137.526,188.185,-62.373,-178.306,7.410,148.905
C03623=1137.522,188.434,-62.395,-178.303,7.413,148.905
C03624=1137.517,188.683,-62.419,-178.300,7.416,148.905
C03625=1137.513,188.932,-62.442,-178.298,7.418,148.905
C03626=1137.508,189.181,-62.466,-178.295,7.420,148.904
C03627=1137.503,189.430,-62.489,-178.292,7.422,148.904
C03628=1137.499,189.679,-62.513,-178.289,7.425,148.904
C03629=1137.494,189.927,-62.537,-178.286,7.428,148.904
C03630=1137.490,190.176,-62.560,-178.284,7.429,148.903
C03631=1137.485,190.425,-62.584,-178.281,7.432,148.903
C03632=1137.480,190.674,-62.608,-178.277,7.435,148.903
C03633=1137.476,190.924,-62.632,-178.275,7.437,148.903
C03634=1137.471,191.172,-62.656,-178.272,7.440,148.902
C03635=1137.467,191.421,-62.679,-178.270,7.442,148.902
C03636=1137.462,191.670,-62.703,-178.266,7.444,148.902
C03637=1137.458,191.918,-62.727,-178.264,7.447,148.902
C03638=1137.453,192.168,-62.750,-178.261,7.449,148.901
C03639=1137.448,192.416,-62.774,-178.258,7.452,148.901
C03640=1137.444,192.665,-62.798,-178.255,7.454,148.901
C03641=1137.439,192.913,-62.822,-178.253,7.456,148.901
C03642=1137.435,193.162,-62.845,-178.249,7.459,148.901
C03643=1137.430,193.411,-62.869,-178.246,7.462,148.900
C03644=1137.425,193.660,-62.893,-178.244,7.464,148.900
C03645=1137.420,193.909,-62.917,-178.241,7.466,148.900
C03646=1137.416,194.158,-62.941,-178.238,7.469,148.900
C03647=1137.412,194.407,-62.965,-178.235,7.471,148.899
C03648=1137.408,194.655,-62.989,-178.233,7.474,148.899
C03649=1137.403,194.904,-63.012,-178.229,7.476,148.899
C03650=1137.398,195.153,-63.037,-178.227,7.479,148.899
C03651=1137.393,195.402,-63.060,-178.224,7.481,148.899
